(* IEC 61131-3 sources: AXOpen/src/components.keyence.vision/ctrl/src/Axo_IV3, 1 file *)

(* ---- Axo_IV3.st ---- *)
USING AXOpen.Core;
USING AXOpen.Messaging;
USING AXOpen.Messaging.Static;
USING AXOpen.Components.Abstractions;
USING Siemens.Simatic.Hardware.Utilities;

NAMESPACE AXOpen.Components.Keyence.Vision
    {S7.extern=ReadWrite}
    {#ix-prop: public string DeviceIpAddress}
    {#ix-prop: public string Proxy}
    CLASS Axo_IV3 EXTENDS AXOpen.Core.AxoComponent
        VAR PUBLIC // HEADER
            {#ix-attr:[Container(Layout.Wrap)]}
            {#ix-attr:[ComponentHeader()]}
            {#ix-set:AttributeName = "<#Progress#>"}
            Progress : INT;
        END_VAR

        VAR PUBLIC // TASKS
            {#ix-attr:[Container(Layout.Wrap)]}
            {#ix-attr:[ComponentDetails("Tasks")]}
            {#ix-set:AttributeName = "<#TriggerTask#>"}
            TriggerTask : AXOpen.Core.AxoTask;
            {#ix-attr:[Container(Layout.Wrap)]}
            {#ix-attr:[ComponentDetails("Tasks")]}
            {#ix-set:AttributeName = "<#Restore#>"}
            RestoreTask : AXOpen.Core.AxoTask;

            {#ix-attr:[Group(GroupLayout.GroupBox)]}
            {#ix-attr:[ComponentDetails("Tasks")]}
            {#ix-set:AttributeName = "<#Required program number#>"}
            RequiredProgramNumber : UINT;
            {#ix-attr:[ComponentDetails("Tasks")]}
            {#ix-set:AttributeName = "<#ChangeProgramTask#>"}
            ChangeProgramTask : AXOpen.Core.AxoTask;
        END_VAR

        VAR PUBLIC // CONFIG
            {#ix-attr:[Container(Layout.Stack)]}
            {#ix-attr:[ComponentDetails("Config")]}
            {#ix-attr:[ReadOnly()]}
            Config  :   Axo_IV3_Config;
        END_VAR

        VAR PUBLIC // STATUS
            {#ix-attr:[Container(Layout.Stack)]}
            {#ix-attr:[ComponentDetails("Status")]}
            {#ix-attr:[ReadOnly()]}
            Status              :   Axo_IV3_Component_Status;
            Messenger           :   AXOpen.Messaging.Static.AxoMessenger;
            TaskMessenger       :   AXOpen.Messaging.Static.AxoMessenger;
        END_VAR

        VAR PUBLIC // HARDWARE SIGNALS
            {#ix-attr:[ComponentDetails("HARDWARE SIGNALS")]}
            {#ix-attr:[Container(Layout.Wrap)]}
            {#ix-attr:[Group(GroupLayout.GroupBox)]}
            {#ix-set:AttributeName = "<#Inputs#>"}
            {#ix-attr:[ReadOnly()]}
            Inputs              :  Axo_IV3_In;
            {#ix-attr:[ComponentDetails("HARDWARE SIGNALS")]}
            {#ix-attr:[Container(Layout.Wrap)]}
            {#ix-attr:[Group(GroupLayout.GroupBox)]}
            {#ix-set:AttributeName = "<#Outputs#>"}
            {#ix-attr:[ReadOnly()]}
            Outputs              :   Axo_IV3_Out;
        END_VAR

        VAR PUBLIC // HARDWARE DIAGNOSTICS TASK
            {#ix-attr:[Container(Layout.Stack)]}
            {#ix-attr:[ComponentDetails("Hardware diagnostics")]}
            {#ix-set:AttributeName = "<#Update diagnostics#>"}
            HardwareDiagnosticsTask :   AXOpen.Io.AxoHardwareDiagnostics;

            LastProgressRoot : ARRAY[0..20] OF INT;
            ProgressRoot : ARRAY[0..20] OF INT;
            ActiveProgressRootIndex : INT;
        END_VAR

        VAR PRIVATE
            _progress       :   INT;
            _infoTimer      :   AXOpen.Timers.OnDelayTimer;
            _errorTimer     :   AXOpen.Timers.OnDelayTimer;
            _data_in        :   ARRAY[0..27] OF BYTE;
            _data_out_12    :   ARRAY[0..11] OF BYTE;
            _word           :   WORD;
            _dword          :   DWORD;

            _initHwCheckDone        :   BOOL;
            _retval                 :   WORD;
            _geoAddr                :   GeoAddr;
            _outHwid                :   UINT;
            _blink                  :   AXOpen.Timers.AxoBlinker;
            _inputsAddress          :   UDINT;
            _inputsCount            :   UINT;
            _outputsAddress         :   UDINT;
            _outputsCount           :   UINT;
            _resultUpdateComplete   :   BOOL;
            _resultNo               :   UINT;
            _programNumber          :   UINT;
            _ProgChangeInterrupted  :   BOOL;
        END_VAR

        METHOD AddProgressToRoot
            VAR_INPUT
                inProgress : INT;
            END_VAR

            var
                lastProgress : INT;
            end_var;

            lastProgress := ProgressRoot[ActiveProgressRootIndex];

            IF inProgress <> lastProgress THEN
                ActiveProgressRootIndex := ActiveProgressRootIndex + 1;
                IF ActiveProgressRootIndex > 20 THEN
                    ActiveProgressRootIndex := 0;
                END_IF;
                ProgressRoot[ActiveProgressRootIndex] := inProgress;
            END_IF;

        END_METHOD

        METHOD ClearProgressRoot
           var
            iterator : INT;
           end_var;

           ActiveProgressRootIndex := 0;
           FOR iterator := 0 TO 20 DO
            LastProgressRoot[iterator] := ProgressRoot[iterator];
                ProgressRoot[iterator] := -1;
           END_FOR;
        END_METHOD

        ///<summary>
        /// Runs tasks and logic of this component.
        /// >[!IMPORTANT] This method must or one of its overloads be called cyclically.
        ///</summary>
        METHOD PUBLIC Run
            VAR_INPUT
                inParent      :   IAxoObject;
                hwID        :   UINT;
            END_VAR

            SUPER.Run(inParent);

            Messenger.Serve(THIS);

            Progress := _progress;

            IF NOT _initHwCheckDone THEN
                IF inParent = NULL THEN
                    Messenger.Activate(UINT#700, eAxoMessageCategory#ProgrammingError);
                    Status.Error.Id := UINT#700;
                    RETURN;
                END_IF;
                IF hwID = UINT#0 THEN
                    Messenger.Activate(UINT#701, eAxoMessageCategory#ProgrammingError);
                    Status.Error.Id := UINT#701;
                    RETURN;
                END_IF;

                Config.HWIDs.HW_Device := hwID;
                _retval := ReadSlotFromHardwareID(hardwareID := Config.HWIDs.HW_Device, geoAddr :=_geoAddr);
                IF _retval = WORD#8090 THEN
                    Messenger.Activate(UINT#702,eAxoMessageCategory#Error);
                    Status.Error.Id := UINT#702;
                    RETURN;
                END_IF;

                //******************Slot 1*****************//
                _geoAddr.Slot   :=  UINT#1;
                _geoAddr.HardwareType := UINT#4; // (4-Module)
                _retval := ReadHardwareIDFromSlot(geoAddr := _geoAddr, hardwareID => Config.HWIDs.HwID_CommandControl);
                IF Config.HWIDs.HwID_CommandControl = UINT#0 THEN
                    Messenger.Activate(UINT#710,eAxoMessageCategory#Error);
                    Status.Error.Id := UINT#710;
                    RETURN;
                END_IF;
                IF _retval = WORD#8091 THEN
                    Messenger.Activate(UINT#711,eAxoMessageCategory#Error);
                    Status.Error.Id := UINT#711;
                    RETURN;
                END_IF;
                IF _retval = WORD#8094 THEN
                    Messenger.Activate(UINT#712,eAxoMessageCategory#Error);
                    Status.Error.Id := UINT#712;
                    RETURN;
                END_IF;
                IF _retval = WORD#8095 THEN
                    Messenger.Activate(UINT#713,eAxoMessageCategory#Error);
                    Status.Error.Id := UINT#713;
                    RETURN;
                END_IF;
                IF _retval = WORD#8096 THEN
                    Messenger.Activate(UINT#714,eAxoMessageCategory#Error);
                    Status.Error.Id := UINT#714;
                    RETURN;
                END_IF;
                IF _retval = WORD#8097 THEN
                    Messenger.Activate(UINT#715,eAxoMessageCategory#Error);
                    Status.Error.Id := UINT#715;
                    RETURN;
                END_IF;
                ReadHardwareIOAddress(hardwareID := (Config.HWIDs.HwID_CommandControl) , inputStartAddress => _inputsAddress , inputCount => _inputsCount , outputStartAddress => _outputsAddress , outputCount => _outputsCount);
                IF _inputsCount <> UINT#0 OR _outputsCount <> UINT#12 THEN
                    Messenger.Activate(UINT#716,eAxoMessageCategory#Error);
                    Status.Error.Id := UINT#716;
                    RETURN;
                END_IF;
                //******************Slot 2*****************//
                _geoAddr.Slot   :=  UINT#2;
                _geoAddr.HardwareType := UINT#4; // (4-Module)
                _retval := ReadHardwareIDFromSlot(geoAddr := _geoAddr, hardwareID => Config.HWIDs.HwID_CommandStatusBits);
                IF Config.HWIDs.HwID_CommandStatusBits = UINT#0 THEN
                    Messenger.Activate(UINT#720,eAxoMessageCategory#Error);
                    Status.Error.Id := UINT#720;
                    RETURN;
                END_IF;
                IF _retval = WORD#8091 THEN
                    Messenger.Activate(UINT#721,eAxoMessageCategory#Error);
                    Status.Error.Id := UINT#721;
                    RETURN;
                END_IF;
                IF _retval = WORD#8094 THEN
                    Messenger.Activate(UINT#722,eAxoMessageCategory#Error);
                    Status.Error.Id := UINT#722;
                    RETURN;
                END_IF;
                IF _retval = WORD#8095 THEN
                    Messenger.Activate(UINT#723,eAxoMessageCategory#Error);
                    Status.Error.Id := UINT#723;
                    RETURN;
                END_IF;
                IF _retval = WORD#8096 THEN
                    Messenger.Activate(UINT#724,eAxoMessageCategory#Error);
                    Status.Error.Id := UINT#724;
                    RETURN;
                END_IF;
                IF _retval = WORD#8097 THEN
                    Messenger.Activate(UINT#725,eAxoMessageCategory#Error);
                    Status.Error.Id := UINT#725;
                    RETURN;
                END_IF;
                ReadHardwareIOAddress(hardwareID := (Config.HWIDs.HwID_CommandStatusBits) , inputStartAddress => _inputsAddress , inputCount => _inputsCount , outputStartAddress => _outputsAddress , outputCount => _outputsCount);
                IF _inputsCount <> UINT#4 OR _outputsCount <> UINT#0 THEN
                    Messenger.Activate(UINT#726,eAxoMessageCategory#Error);
                    Status.Error.Id := UINT#726;
                    RETURN;
                END_IF;
                //******************Slot 3*****************//
                _geoAddr.Slot   :=  UINT#3;
                _geoAddr.HardwareType := UINT#4; // (4-Module)
                _retval := ReadHardwareIDFromSlot(geoAddr := _geoAddr, hardwareID => Config.HWIDs.HwID_DeviceResultBits_1);
                IF Config.HWIDs.HwID_DeviceResultBits_1 = UINT#0 THEN
                    Messenger.Activate(UINT#730,eAxoMessageCategory#Error);
                    Status.Error.Id := UINT#730;
                    RETURN;
                END_IF;
                IF _retval = WORD#8091 THEN
                    Messenger.Activate(UINT#731,eAxoMessageCategory#Error);
                    Status.Error.Id := UINT#731;
                    RETURN;
                END_IF;
                IF _retval = WORD#8094 THEN
                    Messenger.Activate(UINT#732,eAxoMessageCategory#Error);
                    Status.Error.Id := UINT#732;
                    RETURN;
                END_IF;
                IF _retval = WORD#8095 THEN
                    Messenger.Activate(UINT#733,eAxoMessageCategory#Error);
                    Status.Error.Id := UINT#733;
                    RETURN;
                END_IF;
                IF _retval = WORD#8096 THEN
                    Messenger.Activate(UINT#734,eAxoMessageCategory#Error);
                    Status.Error.Id := UINT#734;
                    RETURN;
                END_IF;
                IF _retval = WORD#8097 THEN
                    Messenger.Activate(UINT#735,eAxoMessageCategory#Error);
                    Status.Error.Id := UINT#735;
                    RETURN;
                END_IF;
                ReadHardwareIOAddress(hardwareID := (Config.HWIDs.HwID_DeviceResultBits_1) , inputStartAddress => _inputsAddress , inputCount => _inputsCount , outputStartAddress => _outputsAddress , outputCount => _outputsCount);
                IF _inputsCount <> UINT#4 OR _outputsCount <> UINT#0 THEN
                    Messenger.Activate(UINT#736,eAxoMessageCategory#Error);
                    Status.Error.Id := UINT#736;
                    RETURN;
                END_IF;
                //******************Slot 4*****************//
                _geoAddr.Slot   :=  UINT#4;
                _geoAddr.HardwareType := UINT#4; // (4-Module)
                _retval := ReadHardwareIDFromSlot(geoAddr := _geoAddr, hardwareID => Config.HWIDs.HwID_DeviceStatusWords);
                IF Config.HWIDs.HwID_DeviceStatusWords = UINT#0 THEN
                    Messenger.Activate(UINT#740,eAxoMessageCategory#Error);
                    Status.Error.Id := UINT#740;
                    RETURN;
                END_IF;
                IF _retval = WORD#8091 THEN
                    Messenger.Activate(UINT#741,eAxoMessageCategory#Error);
                    Status.Error.Id := UINT#741;
                    RETURN;
                END_IF;
                IF _retval = WORD#8094 THEN
                    Messenger.Activate(UINT#742,eAxoMessageCategory#Error);
                    Status.Error.Id := UINT#742;
                    RETURN;
                END_IF;
                IF _retval = WORD#8095 THEN
                    Messenger.Activate(UINT#743,eAxoMessageCategory#Error);
                    Status.Error.Id := UINT#743;
                    RETURN;
                END_IF;
                IF _retval = WORD#8096 THEN
                    Messenger.Activate(UINT#744,eAxoMessageCategory#Error);
                    Status.Error.Id := UINT#744;
                    RETURN;
                END_IF;
                IF _retval = WORD#8097 THEN
                    Messenger.Activate(UINT#745,eAxoMessageCategory#Error);
                    Status.Error.Id := UINT#745;
                    RETURN;
                END_IF;
                ReadHardwareIOAddress(hardwareID := (Config.HWIDs.HwID_DeviceStatusWords) , inputStartAddress => _inputsAddress , inputCount => _inputsCount , outputStartAddress => _outputsAddress , outputCount => _outputsCount);
                IF _inputsCount <> UINT#16 OR _outputsCount <> UINT#0 THEN
                    Messenger.Activate(UINT#746,eAxoMessageCategory#Error);
                    Status.Error.Id := UINT#746;
                    RETURN;
                END_IF;
                //******************Slot 5*****************//
                _geoAddr.Slot   :=  UINT#5;
                _geoAddr.HardwareType := UINT#4; // (4-Module)
                _retval := ReadHardwareIDFromSlot(geoAddr := _geoAddr, hardwareID => Config.HWIDs.HwID_DeviceStatistics);
                IF Config.HWIDs.HwID_DeviceStatistics = UINT#0 THEN
                    Messenger.Activate(UINT#750,eAxoMessageCategory#Error);
                    Status.Error.Id := UINT#750;
                    RETURN;
                END_IF;
                IF _retval = WORD#8091 THEN
                    Messenger.Activate(UINT#751,eAxoMessageCategory#Error);
                    Status.Error.Id := UINT#751;
                    RETURN;
                END_IF;
                IF _retval = WORD#8094 THEN
                    Messenger.Activate(UINT#752,eAxoMessageCategory#Error);
                    Status.Error.Id := UINT#752;
                    RETURN;
                END_IF;
                IF _retval = WORD#8095 THEN
                    Messenger.Activate(UINT#753,eAxoMessageCategory#Error);
                    Status.Error.Id := UINT#753;
                    RETURN;
                END_IF;
                IF _retval = WORD#8096 THEN
                    Messenger.Activate(UINT#754,eAxoMessageCategory#Error);
                    Status.Error.Id := UINT#754;
                    RETURN;
                END_IF;
                IF _retval = WORD#8097 THEN
                    Messenger.Activate(UINT#755,eAxoMessageCategory#Error);
                    Status.Error.Id := UINT#755;
                    RETURN;
                END_IF;
                ReadHardwareIOAddress(hardwareID := (Config.HWIDs.HwID_DeviceStatistics) , inputStartAddress => _inputsAddress , inputCount => _inputsCount , outputStartAddress => _outputsAddress , outputCount => _outputsCount);
                IF _inputsCount <> UINT#28 OR _outputsCount <> UINT#0 THEN
                    Messenger.Activate(UINT#756,eAxoMessageCategory#Error);
                    Status.Error.Id := UINT#756;
                    RETURN;
                END_IF;
                //******************Slot 6*****************//
                _geoAddr.Slot   :=  UINT#6;
                _geoAddr.HardwareType := UINT#4; // (4-Module)
                _retval := ReadHardwareIDFromSlot(geoAddr := _geoAddr, hardwareID => Config.HWIDs.HwID_PositionAdjustResult);
                IF Config.HWIDs.HwID_PositionAdjustResult = UINT#0 THEN
                    Messenger.Activate(UINT#760,eAxoMessageCategory#Error);
                    Status.Error.Id := UINT#760;
                    RETURN;
                END_IF;
                IF _retval = WORD#8091 THEN
                    Messenger.Activate(UINT#761,eAxoMessageCategory#Error);
                    Status.Error.Id := UINT#761;
                    RETURN;
                END_IF;
                IF _retval = WORD#8094 THEN
                    Messenger.Activate(UINT#762,eAxoMessageCategory#Error);
                    Status.Error.Id := UINT#762;
                    RETURN;
                END_IF;
                IF _retval = WORD#8095 THEN
                    Messenger.Activate(UINT#763,eAxoMessageCategory#Error);
                    Status.Error.Id := UINT#763;
                    RETURN;
                END_IF;
                IF _retval = WORD#8096 THEN
                    Messenger.Activate(UINT#764,eAxoMessageCategory#Error);
                    Status.Error.Id := UINT#764;
                    RETURN;
                END_IF;
                IF _retval = WORD#8097 THEN
                    Messenger.Activate(UINT#765,eAxoMessageCategory#Error);
                    Status.Error.Id := UINT#765;
                    RETURN;
                END_IF;
                ReadHardwareIOAddress(hardwareID := (Config.HWIDs.HwID_PositionAdjustResult) , inputStartAddress => _inputsAddress , inputCount => _inputsCount , outputStartAddress => _outputsAddress , outputCount => _outputsCount);
                IF _inputsCount <> UINT#20 OR _outputsCount <> UINT#0 THEN
                    Messenger.Activate(UINT#766,eAxoMessageCategory#Error);
                    Status.Error.Id := UINT#766;
                    RETURN;
                END_IF;
                //******************Slot 7*****************//
                _geoAddr.Slot   :=  UINT#7;
                _geoAddr.HardwareType := UINT#4; // (4-Module)
                _retval := ReadHardwareIDFromSlot(geoAddr := _geoAddr, hardwareID => Config.HWIDs.HwID_ToolResult_1);
                IF Config.HWIDs.HwID_ToolResult_1 = UINT#0 THEN
                    Messenger.Activate(UINT#770,eAxoMessageCategory#Error);
                    Status.Error.Id := UINT#770;
                    RETURN;
                END_IF;
                IF _retval = WORD#8091 THEN
                    Messenger.Activate(UINT#771,eAxoMessageCategory#Error);
                    Status.Error.Id := UINT#771;
                    RETURN;
                END_IF;
                IF _retval = WORD#8094 THEN
                    Messenger.Activate(UINT#772,eAxoMessageCategory#Error);
                    Status.Error.Id := UINT#772;
                    RETURN;
                END_IF;
                IF _retval = WORD#8095 THEN
                    Messenger.Activate(UINT#773,eAxoMessageCategory#Error);
                    Status.Error.Id := UINT#773;
                    RETURN;
                END_IF;
                IF _retval = WORD#8096 THEN
                    Messenger.Activate(UINT#774,eAxoMessageCategory#Error);
                    Status.Error.Id := UINT#774;
                    RETURN;
                END_IF;
                IF _retval = WORD#8097 THEN
                    Messenger.Activate(UINT#775,eAxoMessageCategory#Error);
                    Status.Error.Id := UINT#775;
                    RETURN;
                END_IF;
                ReadHardwareIOAddress(hardwareID := (Config.HWIDs.HwID_ToolResult_1) , inputStartAddress => _inputsAddress , inputCount => _inputsCount , outputStartAddress => _outputsAddress , outputCount => _outputsCount);
                IF _inputsCount <> UINT#20 OR _outputsCount <> UINT#0 THEN
                    Messenger.Activate(UINT#776,eAxoMessageCategory#Error);
                    Status.Error.Id := UINT#776;
                    RETURN;
                END_IF;
                //******************Slot 8*****************//
                _geoAddr.Slot   :=  UINT#8;
                _geoAddr.HardwareType := UINT#4; // (4-Module)
                _retval := ReadHardwareIDFromSlot(geoAddr := _geoAddr, hardwareID => Config.HWIDs.HwID_ToolResult_2);
                IF Config.HWIDs.HwID_ToolResult_2 = UINT#0 THEN
                    Messenger.Activate(UINT#780,eAxoMessageCategory#Error);
                    Status.Error.Id := UINT#780;
                    RETURN;
                END_IF;
                IF _retval = WORD#8091 THEN
                    Messenger.Activate(UINT#781,eAxoMessageCategory#Error);
                    Status.Error.Id := UINT#781;
                    RETURN;
                END_IF;
                IF _retval = WORD#8094 THEN
                    Messenger.Activate(UINT#782,eAxoMessageCategory#Error);
                    Status.Error.Id := UINT#782;
                    RETURN;
                END_IF;
                IF _retval = WORD#8095 THEN
                    Messenger.Activate(UINT#783,eAxoMessageCategory#Error);
                    Status.Error.Id := UINT#783;
                    RETURN;
                END_IF;
                IF _retval = WORD#8096 THEN
                    Messenger.Activate(UINT#784,eAxoMessageCategory#Error);
                    Status.Error.Id := UINT#784;
                    RETURN;
                END_IF;
                IF _retval = WORD#8097 THEN
                    Messenger.Activate(UINT#785,eAxoMessageCategory#Error);
                    Status.Error.Id := UINT#785;
                    RETURN;
                END_IF;
                ReadHardwareIOAddress(hardwareID := (Config.HWIDs.HwID_ToolResult_2) , inputStartAddress => _inputsAddress , inputCount => _inputsCount , outputStartAddress => _outputsAddress , outputCount => _outputsCount);
                IF _inputsCount <> UINT#20 OR _outputsCount <> UINT#0 THEN
                    Messenger.Activate(UINT#786,eAxoMessageCategory#Error);
                    Status.Error.Id := UINT#786;
                    RETURN;
                END_IF;
                //******************Slot 9*****************//
                _geoAddr.Slot   :=  UINT#9;
                _geoAddr.HardwareType := UINT#4; // (4-Module)
                _retval := ReadHardwareIDFromSlot(geoAddr := _geoAddr, hardwareID => Config.HWIDs.HwID_ToolResult_3);
                IF Config.HWIDs.HwID_ToolResult_3 = UINT#0 THEN
                    Messenger.Activate(UINT#790,eAxoMessageCategory#Error);
                    Status.Error.Id := UINT#790;
                    RETURN;
                END_IF;
                IF _retval = WORD#8091 THEN
                    Messenger.Activate(UINT#791,eAxoMessageCategory#Error);
                    Status.Error.Id := UINT#791;
                    RETURN;
                END_IF;
                IF _retval = WORD#8094 THEN
                    Messenger.Activate(UINT#792,eAxoMessageCategory#Error);
                    Status.Error.Id := UINT#792;
                    RETURN;
                END_IF;
                IF _retval = WORD#8095 THEN
                    Messenger.Activate(UINT#793,eAxoMessageCategory#Error);
                    Status.Error.Id := UINT#793;
                    RETURN;
                END_IF;
                IF _retval = WORD#8096 THEN
                    Messenger.Activate(UINT#794,eAxoMessageCategory#Error);
                    Status.Error.Id := UINT#794;
                    RETURN;
                END_IF;
                IF _retval = WORD#8097 THEN
                    Messenger.Activate(UINT#795,eAxoMessageCategory#Error);
                    Status.Error.Id := UINT#795;
                    RETURN;
                END_IF;
                ReadHardwareIOAddress(hardwareID := (Config.HWIDs.HwID_ToolResult_3) , inputStartAddress => _inputsAddress , inputCount => _inputsCount , outputStartAddress => _outputsAddress , outputCount => _outputsCount);
                IF _inputsCount <> UINT#20 OR _outputsCount <> UINT#0 THEN
                    Messenger.Activate(UINT#796,eAxoMessageCategory#Error);
                    Status.Error.Id := UINT#796;
                    RETURN;
                END_IF;
                //******************Slot 10*****************//
                _geoAddr.Slot   :=  UINT#10;
                _geoAddr.HardwareType := UINT#4; // (4-Module)
                _retval := ReadHardwareIDFromSlot(geoAddr := _geoAddr, hardwareID => Config.HWIDs.HwID_ToolResult_4);
                IF Config.HWIDs.HwID_ToolResult_4 = UINT#0 THEN
                    Messenger.Activate(UINT#800,eAxoMessageCategory#Error);
                    Status.Error.Id := UINT#800;
                    RETURN;
                END_IF;
                IF _retval = WORD#8091 THEN
                    Messenger.Activate(UINT#801,eAxoMessageCategory#Error);
                    Status.Error.Id := UINT#801;
                    RETURN;
                END_IF;
                IF _retval = WORD#8094 THEN
                    Messenger.Activate(UINT#802,eAxoMessageCategory#Error);
                    Status.Error.Id := UINT#802;
                    RETURN;
                END_IF;
                IF _retval = WORD#8095 THEN
                    Messenger.Activate(UINT#803,eAxoMessageCategory#Error);
                    Status.Error.Id := UINT#803;
                    RETURN;
                END_IF;
                IF _retval = WORD#8096 THEN
                    Messenger.Activate(UINT#804,eAxoMessageCategory#Error);
                    Status.Error.Id := UINT#804;
                    RETURN;
                END_IF;
                IF _retval = WORD#8097 THEN
                    Messenger.Activate(UINT#805,eAxoMessageCategory#Error);
                    Status.Error.Id := UINT#805;
                    RETURN;
                END_IF;
                ReadHardwareIOAddress(hardwareID := (Config.HWIDs.HwID_ToolResult_4) , inputStartAddress => _inputsAddress , inputCount => _inputsCount , outputStartAddress => _outputsAddress , outputCount => _outputsCount);
                IF _inputsCount <> UINT#20 OR _outputsCount <> UINT#0 THEN
                    Messenger.Activate(UINT#806,eAxoMessageCategory#Error);
                    Status.Error.Id := UINT#806;
                    RETURN;
                END_IF;
                //******************Slot 11*****************//
                _geoAddr.Slot   :=  UINT#11;
                _geoAddr.HardwareType := UINT#4; // (4-Module)
                _retval := ReadHardwareIDFromSlot(geoAddr := _geoAddr, hardwareID => Config.HWIDs.HwID_ToolResult_5);
                IF Config.HWIDs.HwID_ToolResult_5 = UINT#0 THEN
                    Messenger.Activate(UINT#810,eAxoMessageCategory#Error);
                    Status.Error.Id := UINT#810;
                    RETURN;
                END_IF;
                IF _retval = WORD#8091 THEN
                    Messenger.Activate(UINT#811,eAxoMessageCategory#Error);
                    Status.Error.Id := UINT#811;
                    RETURN;
                END_IF;
                IF _retval = WORD#8094 THEN
                    Messenger.Activate(UINT#812,eAxoMessageCategory#Error);
                    Status.Error.Id := UINT#812;
                    RETURN;
                END_IF;
                IF _retval = WORD#8095 THEN
                    Messenger.Activate(UINT#813,eAxoMessageCategory#Error);
                    Status.Error.Id := UINT#813;
                    RETURN;
                END_IF;
                IF _retval = WORD#8096 THEN
                    Messenger.Activate(UINT#814,eAxoMessageCategory#Error);
                    Status.Error.Id := UINT#814;
                    RETURN;
                END_IF;
                IF _retval = WORD#8097 THEN
                    Messenger.Activate(UINT#815,eAxoMessageCategory#Error);
                    Status.Error.Id := UINT#815;
                    RETURN;
                END_IF;
                ReadHardwareIOAddress(hardwareID := (Config.HWIDs.HwID_ToolResult_5) , inputStartAddress => _inputsAddress , inputCount => _inputsCount , outputStartAddress => _outputsAddress , outputCount => _outputsCount);
                IF _inputsCount <> UINT#20 OR _outputsCount <> UINT#0 THEN
                    Messenger.Activate(UINT#816,eAxoMessageCategory#Error);
                    Status.Error.Id := UINT#816;
                    RETURN;
                END_IF;
                //******************Slot 12*****************//
                _geoAddr.Slot   :=  UINT#12;
                _geoAddr.HardwareType := UINT#4; // (4-Module)
                _retval := ReadHardwareIDFromSlot(geoAddr := _geoAddr, hardwareID => Config.HWIDs.HwID_ToolResult_6);
                IF Config.HWIDs.HwID_ToolResult_6 = UINT#0 THEN
                    Messenger.Activate(UINT#820,eAxoMessageCategory#Error);
                    Status.Error.Id := UINT#820;
                    RETURN;
                END_IF;
                IF _retval = WORD#8091 THEN
                    Messenger.Activate(UINT#821,eAxoMessageCategory#Error);
                    Status.Error.Id := UINT#821;
                    RETURN;
                END_IF;
                IF _retval = WORD#8094 THEN
                    Messenger.Activate(UINT#822,eAxoMessageCategory#Error);
                    Status.Error.Id := UINT#822;
                    RETURN;
                END_IF;
                IF _retval = WORD#8095 THEN
                    Messenger.Activate(UINT#823,eAxoMessageCategory#Error);
                    Status.Error.Id := UINT#823;
                    RETURN;
                END_IF;
                IF _retval = WORD#8096 THEN
                    Messenger.Activate(UINT#824,eAxoMessageCategory#Error);
                    Status.Error.Id := UINT#824;
                    RETURN;
                END_IF;
                IF _retval = WORD#8097 THEN
                    Messenger.Activate(UINT#825,eAxoMessageCategory#Error);
                    Status.Error.Id := UINT#825;
                    RETURN;
                END_IF;
                ReadHardwareIOAddress(hardwareID := (Config.HWIDs.HwID_ToolResult_6) , inputStartAddress => _inputsAddress , inputCount => _inputsCount , outputStartAddress => _outputsAddress , outputCount => _outputsCount);
                IF _inputsCount <> UINT#20 OR _outputsCount <> UINT#0 THEN
                    Messenger.Activate(UINT#826,eAxoMessageCategory#Error);
                    Status.Error.Id := UINT#826;
                    RETURN;
                END_IF;
                //******************Slot 13*****************//
                _geoAddr.Slot   :=  UINT#13;
                _geoAddr.HardwareType := UINT#4; // (4-Module)
                _retval := ReadHardwareIDFromSlot(geoAddr := _geoAddr, hardwareID => Config.HWIDs.HwID_ToolResult_7);
                IF Config.HWIDs.HwID_ToolResult_7 = UINT#0 THEN
                    Messenger.Activate(UINT#830,eAxoMessageCategory#Error);
                    Status.Error.Id := UINT#830;
                    RETURN;
                END_IF;
                IF _retval = WORD#8091 THEN
                    Messenger.Activate(UINT#831,eAxoMessageCategory#Error);
                    Status.Error.Id := UINT#831;
                    RETURN;
                END_IF;
                IF _retval = WORD#8094 THEN
                    Messenger.Activate(UINT#832,eAxoMessageCategory#Error);
                    Status.Error.Id := UINT#832;
                    RETURN;
                END_IF;
                IF _retval = WORD#8095 THEN
                    Messenger.Activate(UINT#833,eAxoMessageCategory#Error);
                    Status.Error.Id := UINT#833;
                    RETURN;
                END_IF;
                IF _retval = WORD#8096 THEN
                    Messenger.Activate(UINT#834,eAxoMessageCategory#Error);
                    Status.Error.Id := UINT#834;
                    RETURN;
                END_IF;
                IF _retval = WORD#8097 THEN
                    Messenger.Activate(UINT#835,eAxoMessageCategory#Error);
                    Status.Error.Id := UINT#835;
                    RETURN;
                END_IF;
                ReadHardwareIOAddress(hardwareID := (Config.HWIDs.HwID_ToolResult_7) , inputStartAddress => _inputsAddress , inputCount => _inputsCount , outputStartAddress => _outputsAddress , outputCount => _outputsCount);
                IF _inputsCount <> UINT#20 OR _outputsCount <> UINT#0 THEN
                    Messenger.Activate(UINT#836,eAxoMessageCategory#Error);
                    Status.Error.Id := UINT#836;
                    RETURN;
                END_IF;
                //******************Slot 14*****************//
                _geoAddr.Slot   :=  UINT#14;
                _geoAddr.HardwareType := UINT#4; // (4-Module)
                _retval := ReadHardwareIDFromSlot(geoAddr := _geoAddr, hardwareID => Config.HWIDs.HwID_ToolResult_8);
                IF Config.HWIDs.HwID_ToolResult_8 = UINT#0 THEN
                    Messenger.Activate(UINT#840,eAxoMessageCategory#Error);
                    Status.Error.Id := UINT#840;
                    RETURN;
                END_IF;
                IF _retval = WORD#8091 THEN
                    Messenger.Activate(UINT#841,eAxoMessageCategory#Error);
                    Status.Error.Id := UINT#841;
                    RETURN;
                END_IF;
                IF _retval = WORD#8094 THEN
                    Messenger.Activate(UINT#842,eAxoMessageCategory#Error);
                    Status.Error.Id := UINT#842;
                    RETURN;
                END_IF;
                IF _retval = WORD#8095 THEN
                    Messenger.Activate(UINT#843,eAxoMessageCategory#Error);
                    Status.Error.Id := UINT#843;
                    RETURN;
                END_IF;
                IF _retval = WORD#8096 THEN
                    Messenger.Activate(UINT#844,eAxoMessageCategory#Error);
                    Status.Error.Id := UINT#844;
                    RETURN;
                END_IF;
                IF _retval = WORD#8097 THEN
                    Messenger.Activate(UINT#845,eAxoMessageCategory#Error);
                    Status.Error.Id := UINT#845;
                    RETURN;
                END_IF;
                ReadHardwareIOAddress(hardwareID := (Config.HWIDs.HwID_ToolResult_8) , inputStartAddress => _inputsAddress , inputCount => _inputsCount , outputStartAddress => _outputsAddress , outputCount => _outputsCount);
                IF _inputsCount <> UINT#20 OR _outputsCount <> UINT#0 THEN
                    Messenger.Activate(UINT#846,eAxoMessageCategory#Error);
                    Status.Error.Id := UINT#846;
                    RETURN;
                END_IF;
                //******************Slot 15*****************//
                _geoAddr.Slot   :=  UINT#15;
                _geoAddr.HardwareType := UINT#4; // (4-Module)
                _retval := ReadHardwareIDFromSlot(geoAddr := _geoAddr, hardwareID => Config.HWIDs.HwID_ToolResult_9);
                IF Config.HWIDs.HwID_ToolResult_9 = UINT#0 THEN
                    Messenger.Activate(UINT#850,eAxoMessageCategory#Error);
                    Status.Error.Id := UINT#850;
                    RETURN;
                END_IF;
                IF _retval = WORD#8091 THEN
                    Messenger.Activate(UINT#851,eAxoMessageCategory#Error);
                    Status.Error.Id := UINT#851;
                    RETURN;
                END_IF;
                IF _retval = WORD#8094 THEN
                    Messenger.Activate(UINT#852,eAxoMessageCategory#Error);
                    Status.Error.Id := UINT#852;
                    RETURN;
                END_IF;
                IF _retval = WORD#8095 THEN
                    Messenger.Activate(UINT#853,eAxoMessageCategory#Error);
                    Status.Error.Id := UINT#853;
                    RETURN;
                END_IF;
                IF _retval = WORD#8096 THEN
                    Messenger.Activate(UINT#854,eAxoMessageCategory#Error);
                    Status.Error.Id := UINT#854;
                    RETURN;
                END_IF;
                IF _retval = WORD#8097 THEN
                    Messenger.Activate(UINT#855,eAxoMessageCategory#Error);
                    Status.Error.Id := UINT#855;
                    RETURN;
                END_IF;
                ReadHardwareIOAddress(hardwareID := (Config.HWIDs.HwID_ToolResult_9) , inputStartAddress => _inputsAddress , inputCount => _inputsCount , outputStartAddress => _outputsAddress , outputCount => _outputsCount);
                IF _inputsCount <> UINT#20 OR _outputsCount <> UINT#0 THEN
                    Messenger.Activate(UINT#856,eAxoMessageCategory#Error);
                    Status.Error.Id := UINT#856;
                    RETURN;
                END_IF;
                //******************Slot 16*****************//
                _geoAddr.Slot   :=  UINT#16;
                _geoAddr.HardwareType := UINT#4; // (4-Module)
                _retval := ReadHardwareIDFromSlot(geoAddr := _geoAddr, hardwareID => Config.HWIDs.HwID_ToolResult_10);
                IF Config.HWIDs.HwID_ToolResult_10 = UINT#0 THEN
                    Messenger.Activate(UINT#860,eAxoMessageCategory#Error);
                    Status.Error.Id := UINT#860;
                    RETURN;
                END_IF;
                IF _retval = WORD#8091 THEN
                    Messenger.Activate(UINT#861,eAxoMessageCategory#Error);
                    Status.Error.Id := UINT#861;
                    RETURN;
                END_IF;
                IF _retval = WORD#8094 THEN
                    Messenger.Activate(UINT#862,eAxoMessageCategory#Error);
                    Status.Error.Id := UINT#862;
                    RETURN;
                END_IF;
                IF _retval = WORD#8095 THEN
                    Messenger.Activate(UINT#863,eAxoMessageCategory#Error);
                    Status.Error.Id := UINT#863;
                    RETURN;
                END_IF;
                IF _retval = WORD#8096 THEN
                    Messenger.Activate(UINT#864,eAxoMessageCategory#Error);
                    Status.Error.Id := UINT#864;
                    RETURN;
                END_IF;
                IF _retval = WORD#8097 THEN
                    Messenger.Activate(UINT#865,eAxoMessageCategory#Error);
                    Status.Error.Id := UINT#865;
                    RETURN;
                END_IF;
                ReadHardwareIOAddress(hardwareID := (Config.HWIDs.HwID_ToolResult_10) , inputStartAddress => _inputsAddress , inputCount => _inputsCount , outputStartAddress => _outputsAddress , outputCount => _outputsCount);
                IF _inputsCount <> UINT#20 OR _outputsCount <> UINT#0 THEN
                    Messenger.Activate(UINT#866,eAxoMessageCategory#Error);
                    Status.Error.Id := UINT#866;
                    RETURN;
                END_IF;
                //******************Slot 17*****************//
                _geoAddr.Slot   :=  UINT#17;
                _geoAddr.HardwareType := UINT#4; // (4-Module)
                _retval := ReadHardwareIDFromSlot(geoAddr := _geoAddr, hardwareID => Config.HWIDs.HwID_ToolResult_11);
                IF Config.HWIDs.HwID_ToolResult_11 = UINT#0 THEN
                    Messenger.Activate(UINT#870,eAxoMessageCategory#Error);
                    Status.Error.Id := UINT#870;
                    RETURN;
                END_IF;
                IF _retval = WORD#8091 THEN
                    Messenger.Activate(UINT#871,eAxoMessageCategory#Error);
                    Status.Error.Id := UINT#871;
                    RETURN;
                END_IF;
                IF _retval = WORD#8094 THEN
                    Messenger.Activate(UINT#872,eAxoMessageCategory#Error);
                    Status.Error.Id := UINT#872;
                    RETURN;
                END_IF;
                IF _retval = WORD#8095 THEN
                    Messenger.Activate(UINT#873,eAxoMessageCategory#Error);
                    Status.Error.Id := UINT#873;
                    RETURN;
                END_IF;
                IF _retval = WORD#8096 THEN
                    Messenger.Activate(UINT#874,eAxoMessageCategory#Error);
                    Status.Error.Id := UINT#874;
                    RETURN;
                END_IF;
                IF _retval = WORD#8097 THEN
                    Messenger.Activate(UINT#875,eAxoMessageCategory#Error);
                    Status.Error.Id := UINT#875;
                    RETURN;
                END_IF;
                ReadHardwareIOAddress(hardwareID := (Config.HWIDs.HwID_ToolResult_11) , inputStartAddress => _inputsAddress , inputCount => _inputsCount , outputStartAddress => _outputsAddress , outputCount => _outputsCount);
                IF _inputsCount <> UINT#20 OR _outputsCount <> UINT#0 THEN
                    Messenger.Activate(UINT#876,eAxoMessageCategory#Error);
                    Status.Error.Id := UINT#876;
                    RETURN;
                END_IF;
                //******************Slot 18*****************//
                _geoAddr.Slot   :=  UINT#18;
                _geoAddr.HardwareType := UINT#4; // (4-Module)
                _retval := ReadHardwareIDFromSlot(geoAddr := _geoAddr, hardwareID => Config.HWIDs.HwID_ToolResult_12);
                IF Config.HWIDs.HwID_ToolResult_12 = UINT#0 THEN
                    Messenger.Activate(UINT#880,eAxoMessageCategory#Error);
                    Status.Error.Id := UINT#880;
                    RETURN;
                END_IF;
                IF _retval = WORD#8091 THEN
                    Messenger.Activate(UINT#881,eAxoMessageCategory#Error);
                    Status.Error.Id := UINT#881;
                    RETURN;
                END_IF;
                IF _retval = WORD#8094 THEN
                    Messenger.Activate(UINT#882,eAxoMessageCategory#Error);
                    Status.Error.Id := UINT#882;
                    RETURN;
                END_IF;
                IF _retval = WORD#8095 THEN
                    Messenger.Activate(UINT#883,eAxoMessageCategory#Error);
                    Status.Error.Id := UINT#883;
                    RETURN;
                END_IF;
                IF _retval = WORD#8096 THEN
                    Messenger.Activate(UINT#884,eAxoMessageCategory#Error);
                    Status.Error.Id := UINT#884;
                    RETURN;
                END_IF;
                IF _retval = WORD#8097 THEN
                    Messenger.Activate(UINT#885,eAxoMessageCategory#Error);
                    Status.Error.Id := UINT#885;
                    RETURN;
                END_IF;
                ReadHardwareIOAddress(hardwareID := (Config.HWIDs.HwID_ToolResult_12) , inputStartAddress => _inputsAddress , inputCount => _inputsCount , outputStartAddress => _outputsAddress , outputCount => _outputsCount);
                IF _inputsCount <> UINT#20 OR _outputsCount <> UINT#0 THEN
                    Messenger.Activate(UINT#886,eAxoMessageCategory#Error);
                    Status.Error.Id := UINT#886;
                    RETURN;
                END_IF;
                //******************Slot 19*****************//
                _geoAddr.Slot   :=  UINT#19;
                _geoAddr.HardwareType := UINT#4; // (4-Module)
                _retval := ReadHardwareIDFromSlot(geoAddr := _geoAddr, hardwareID => Config.HWIDs.HwID_ToolResult_13);
                IF Config.HWIDs.HwID_ToolResult_13 = UINT#0 THEN
                    Messenger.Activate(UINT#890,eAxoMessageCategory#Error);
                    Status.Error.Id := UINT#890;
                    RETURN;
                END_IF;
                IF _retval = WORD#8091 THEN
                    Messenger.Activate(UINT#891,eAxoMessageCategory#Error);
                    Status.Error.Id := UINT#891;
                    RETURN;
                END_IF;
                IF _retval = WORD#8094 THEN
                    Messenger.Activate(UINT#892,eAxoMessageCategory#Error);
                    Status.Error.Id := UINT#892;
                    RETURN;
                END_IF;
                IF _retval = WORD#8095 THEN
                    Messenger.Activate(UINT#893,eAxoMessageCategory#Error);
                    Status.Error.Id := UINT#893;
                    RETURN;
                END_IF;
                IF _retval = WORD#8096 THEN
                    Messenger.Activate(UINT#894,eAxoMessageCategory#Error);
                    Status.Error.Id := UINT#894;
                    RETURN;
                END_IF;
                IF _retval = WORD#8097 THEN
                    Messenger.Activate(UINT#895,eAxoMessageCategory#Error);
                    Status.Error.Id := UINT#895;
                    RETURN;
                END_IF;
                ReadHardwareIOAddress(hardwareID := (Config.HWIDs.HwID_ToolResult_13) , inputStartAddress => _inputsAddress , inputCount => _inputsCount , outputStartAddress => _outputsAddress , outputCount => _outputsCount);
                IF _inputsCount <> UINT#20 OR _outputsCount <> UINT#0 THEN
                    Messenger.Activate(UINT#896,eAxoMessageCategory#Error);
                    Status.Error.Id := UINT#896;
                    RETURN;
                END_IF;
                //******************Slot 20*****************//
                _geoAddr.Slot   :=  UINT#20;
                _geoAddr.HardwareType := UINT#4; // (4-Module)
                _retval := ReadHardwareIDFromSlot(geoAddr := _geoAddr, hardwareID => Config.HWIDs.HwID_ToolResult_14);
                IF Config.HWIDs.HwID_ToolResult_14 = UINT#0 THEN
                    Messenger.Activate(UINT#900,eAxoMessageCategory#Error);
                    Status.Error.Id := UINT#900;
                    RETURN;
                END_IF;
                IF _retval = WORD#8091 THEN
                    Messenger.Activate(UINT#901,eAxoMessageCategory#Error);
                    Status.Error.Id := UINT#901;
                    RETURN;
                END_IF;
                IF _retval = WORD#8094 THEN
                    Messenger.Activate(UINT#902,eAxoMessageCategory#Error);
                    Status.Error.Id := UINT#902;
                    RETURN;
                END_IF;
                IF _retval = WORD#8095 THEN
                    Messenger.Activate(UINT#903,eAxoMessageCategory#Error);
                    Status.Error.Id := UINT#903;
                    RETURN;
                END_IF;
                IF _retval = WORD#8096 THEN
                    Messenger.Activate(UINT#904,eAxoMessageCategory#Error);
                    Status.Error.Id := UINT#904;
                    RETURN;
                END_IF;
                IF _retval = WORD#8097 THEN
                    Messenger.Activate(UINT#905,eAxoMessageCategory#Error);
                    Status.Error.Id := UINT#905;
                    RETURN;
                END_IF;
                ReadHardwareIOAddress(hardwareID := (Config.HWIDs.HwID_ToolResult_14) , inputStartAddress => _inputsAddress , inputCount => _inputsCount , outputStartAddress => _outputsAddress , outputCount => _outputsCount);
                IF _inputsCount <> UINT#20 OR _outputsCount <> UINT#0 THEN
                    Messenger.Activate(UINT#916,eAxoMessageCategory#Error);
                    Status.Error.Id := UINT#916;
                    RETURN;
                END_IF;
                //******************Slot 21*****************//
                _geoAddr.Slot   :=  UINT#21;
                _geoAddr.HardwareType := UINT#4; // (4-Module)
                _retval := ReadHardwareIDFromSlot(geoAddr := _geoAddr, hardwareID => Config.HWIDs.HwID_ToolResult_15);
                IF Config.HWIDs.HwID_ToolResult_15 = UINT#0 THEN
                    Messenger.Activate(UINT#910,eAxoMessageCategory#Error);
                    Status.Error.Id := UINT#910;
                    RETURN;
                END_IF;
                IF _retval = WORD#8091 THEN
                    Messenger.Activate(UINT#911,eAxoMessageCategory#Error);
                    Status.Error.Id := UINT#911;
                    RETURN;
                END_IF;
                IF _retval = WORD#8094 THEN
                    Messenger.Activate(UINT#912,eAxoMessageCategory#Error);
                    Status.Error.Id := UINT#912;
                    RETURN;
                END_IF;
                IF _retval = WORD#8095 THEN
                    Messenger.Activate(UINT#913,eAxoMessageCategory#Error);
                    Status.Error.Id := UINT#913;
                    RETURN;
                END_IF;
                IF _retval = WORD#8096 THEN
                    Messenger.Activate(UINT#914,eAxoMessageCategory#Error);
                    Status.Error.Id := UINT#914;
                    RETURN;
                END_IF;
                IF _retval = WORD#8097 THEN
                    Messenger.Activate(UINT#715,eAxoMessageCategory#Error);
                    Status.Error.Id := UINT#715;
                    RETURN;
                END_IF;
                ReadHardwareIOAddress(hardwareID := (Config.HWIDs.HwID_ToolResult_15) , inputStartAddress => _inputsAddress , inputCount => _inputsCount , outputStartAddress => _outputsAddress , outputCount => _outputsCount);
                IF _inputsCount <> UINT#20 OR _outputsCount <> UINT#0 THEN
                    Messenger.Activate(UINT#916,eAxoMessageCategory#Error);
                    Status.Error.Id := UINT#916;
                    RETURN;
                END_IF;
                //******************Slot 22*****************//
                _geoAddr.Slot   :=  UINT#22;
                _geoAddr.HardwareType := UINT#4; // (4-Module)
                _retval := ReadHardwareIDFromSlot(geoAddr := _geoAddr, hardwareID => Config.HWIDs.HwID_ToolResult_16);
                IF Config.HWIDs.HwID_ToolResult_16 = UINT#0 THEN
                    Messenger.Activate(UINT#920,eAxoMessageCategory#Error);
                    Status.Error.Id := UINT#920;
                    RETURN;
                END_IF;
                IF _retval = WORD#8091 THEN
                    Messenger.Activate(UINT#921,eAxoMessageCategory#Error);
                    Status.Error.Id := UINT#921;
                    RETURN;
                END_IF;
                IF _retval = WORD#8094 THEN
                    Messenger.Activate(UINT#922,eAxoMessageCategory#Error);
                    Status.Error.Id := UINT#922;
                    RETURN;
                END_IF;
                IF _retval = WORD#8095 THEN
                    Messenger.Activate(UINT#923,eAxoMessageCategory#Error);
                    Status.Error.Id := UINT#923;
                    RETURN;
                END_IF;
                IF _retval = WORD#8096 THEN
                    Messenger.Activate(UINT#924,eAxoMessageCategory#Error);
                    Status.Error.Id := UINT#924;
                    RETURN;
                END_IF;
                IF _retval = WORD#8097 THEN
                    Messenger.Activate(UINT#925,eAxoMessageCategory#Error);
                    Status.Error.Id := UINT#925;
                    RETURN;
                END_IF;
                ReadHardwareIOAddress(hardwareID := (Config.HWIDs.HwID_ToolResult_16) , inputStartAddress => _inputsAddress , inputCount => _inputsCount , outputStartAddress => _outputsAddress , outputCount => _outputsCount);
                IF _inputsCount <> UINT#20 OR _outputsCount <> UINT#0 THEN
                    Messenger.Activate(UINT#926,eAxoMessageCategory#Error);
                    Status.Error.Id := UINT#926;
                    RETURN;
                END_IF;
                //******************Slot 23*****************//
                _geoAddr.Slot   :=  UINT#23;
                _geoAddr.HardwareType := UINT#4; // (4-Module)
                _retval := ReadHardwareIDFromSlot(geoAddr := _geoAddr, hardwareID => Config.HWIDs.HwID_ToolResult_17);
                IF Config.HWIDs.HwID_ToolResult_17 = UINT#0 THEN
                    Messenger.Activate(UINT#930,eAxoMessageCategory#Error);
                    Status.Error.Id := UINT#930;
                    RETURN;
                END_IF;
                IF _retval = WORD#8091 THEN
                    Messenger.Activate(UINT#931,eAxoMessageCategory#Error);
                    Status.Error.Id := UINT#931;
                    RETURN;
                END_IF;
                IF _retval = WORD#8094 THEN
                    Messenger.Activate(UINT#932,eAxoMessageCategory#Error);
                    Status.Error.Id := UINT#932;
                    RETURN;
                END_IF;
                IF _retval = WORD#8095 THEN
                    Messenger.Activate(UINT#933,eAxoMessageCategory#Error);
                    Status.Error.Id := UINT#933;
                    RETURN;
                END_IF;
                IF _retval = WORD#8096 THEN
                    Messenger.Activate(UINT#934,eAxoMessageCategory#Error);
                    Status.Error.Id := UINT#934;
                    RETURN;
                END_IF;
                IF _retval = WORD#8097 THEN
                    Messenger.Activate(UINT#935,eAxoMessageCategory#Error);
                    Status.Error.Id := UINT#935;
                    RETURN;
                END_IF;
                ReadHardwareIOAddress(hardwareID := (Config.HWIDs.HwID_ToolResult_17) , inputStartAddress => _inputsAddress , inputCount => _inputsCount , outputStartAddress => _outputsAddress , outputCount => _outputsCount);
                IF _inputsCount <> UINT#20 OR _outputsCount <> UINT#0 THEN
                    Messenger.Activate(UINT#936,eAxoMessageCategory#Error);
                    Status.Error.Id := UINT#936;
                    RETURN;
                END_IF;
                //******************Slot 24*****************//
                _geoAddr.Slot   :=  UINT#24;
                _geoAddr.HardwareType := UINT#4; // (4-Module)
                _retval := ReadHardwareIDFromSlot(geoAddr := _geoAddr, hardwareID => Config.HWIDs.HwID_ToolResult_18);
                IF Config.HWIDs.HwID_ToolResult_18 = UINT#0 THEN
                    Messenger.Activate(UINT#940,eAxoMessageCategory#Error);
                    Status.Error.Id := UINT#940;
                    RETURN;
                END_IF;
                IF _retval = WORD#8091 THEN
                    Messenger.Activate(UINT#941,eAxoMessageCategory#Error);
                    Status.Error.Id := UINT#941;
                    RETURN;
                END_IF;
                IF _retval = WORD#8094 THEN
                    Messenger.Activate(UINT#942,eAxoMessageCategory#Error);
                    Status.Error.Id := UINT#942;
                    RETURN;
                END_IF;
                IF _retval = WORD#8095 THEN
                    Messenger.Activate(UINT#943,eAxoMessageCategory#Error);
                    Status.Error.Id := UINT#943;
                    RETURN;
                END_IF;
                IF _retval = WORD#8096 THEN
                    Messenger.Activate(UINT#944,eAxoMessageCategory#Error);
                    Status.Error.Id := UINT#944;
                    RETURN;
                END_IF;
                IF _retval = WORD#8097 THEN
                    Messenger.Activate(UINT#945,eAxoMessageCategory#Error);
                    Status.Error.Id := UINT#945;
                    RETURN;
                END_IF;
                ReadHardwareIOAddress(hardwareID := (Config.HWIDs.HwID_ToolResult_18) , inputStartAddress => _inputsAddress , inputCount => _inputsCount , outputStartAddress => _outputsAddress , outputCount => _outputsCount);
                IF _inputsCount <> UINT#20 OR _outputsCount <> UINT#0 THEN
                    Messenger.Activate(UINT#946,eAxoMessageCategory#Error);
                    Status.Error.Id := UINT#946;
                    RETURN;
                END_IF;
                //******************Slot 25*****************//
                _geoAddr.Slot   :=  UINT#25;
                _geoAddr.HardwareType := UINT#4; // (4-Module)
                _retval := ReadHardwareIDFromSlot(geoAddr := _geoAddr, hardwareID => Config.HWIDs.HwID_ToolResult_19);
                IF Config.HWIDs.HwID_ToolResult_19 = UINT#0 THEN
                    Messenger.Activate(UINT#950,eAxoMessageCategory#Error);
                    Status.Error.Id := UINT#950;
                    RETURN;
                END_IF;
                IF _retval = WORD#8091 THEN
                    Messenger.Activate(UINT#951,eAxoMessageCategory#Error);
                    Status.Error.Id := UINT#951;
                    RETURN;
                END_IF;
                IF _retval = WORD#8094 THEN
                    Messenger.Activate(UINT#952,eAxoMessageCategory#Error);
                    Status.Error.Id := UINT#952;
                    RETURN;
                END_IF;
                IF _retval = WORD#8095 THEN
                    Messenger.Activate(UINT#953,eAxoMessageCategory#Error);
                    Status.Error.Id := UINT#953;
                    RETURN;
                END_IF;
                IF _retval = WORD#8096 THEN
                    Messenger.Activate(UINT#954,eAxoMessageCategory#Error);
                    Status.Error.Id := UINT#954;
                    RETURN;
                END_IF;
                IF _retval = WORD#8097 THEN
                    Messenger.Activate(UINT#955,eAxoMessageCategory#Error);
                    Status.Error.Id := UINT#955;
                    RETURN;
                END_IF;
                ReadHardwareIOAddress(hardwareID := (Config.HWIDs.HwID_ToolResult_19) , inputStartAddress => _inputsAddress , inputCount => _inputsCount , outputStartAddress => _outputsAddress , outputCount => _outputsCount);
                IF _inputsCount <> UINT#20 OR _outputsCount <> UINT#0 THEN
                    Messenger.Activate(UINT#956,eAxoMessageCategory#Error);
                    Status.Error.Id := UINT#956;
                    RETURN;
                END_IF;
                //******************Slot 26*****************//
                _geoAddr.Slot   :=  UINT#26;
                _geoAddr.HardwareType := UINT#4; // (4-Module)
                _retval := ReadHardwareIDFromSlot(geoAddr := _geoAddr, hardwareID => Config.HWIDs.HwID_ToolResult_20);
                IF Config.HWIDs.HwID_ToolResult_20 = UINT#0 THEN
                    Messenger.Activate(UINT#960,eAxoMessageCategory#Error);
                    Status.Error.Id := UINT#960;
                    RETURN;
                END_IF;
                IF _retval = WORD#8091 THEN
                    Messenger.Activate(UINT#961,eAxoMessageCategory#Error);
                    Status.Error.Id := UINT#961;
                    RETURN;
                END_IF;
                IF _retval = WORD#8094 THEN
                    Messenger.Activate(UINT#962,eAxoMessageCategory#Error);
                    Status.Error.Id := UINT#962;
                    RETURN;
                END_IF;
                IF _retval = WORD#8095 THEN
                    Messenger.Activate(UINT#963,eAxoMessageCategory#Error);
                    Status.Error.Id := UINT#963;
                    RETURN;
                END_IF;
                IF _retval = WORD#8096 THEN
                    Messenger.Activate(UINT#964,eAxoMessageCategory#Error);
                    Status.Error.Id := UINT#964;
                    RETURN;
                END_IF;
                IF _retval = WORD#8097 THEN
                    Messenger.Activate(UINT#965,eAxoMessageCategory#Error);
                    Status.Error.Id := UINT#965;
                    RETURN;
                END_IF;
                ReadHardwareIOAddress(hardwareID := (Config.HWIDs.HwID_ToolResult_20) , inputStartAddress => _inputsAddress , inputCount => _inputsCount , outputStartAddress => _outputsAddress , outputCount => _outputsCount);
                IF _inputsCount <> UINT#20 OR _outputsCount <> UINT#0 THEN
                    Messenger.Activate(UINT#966,eAxoMessageCategory#Error);
                    Status.Error.Id := UINT#966;
                    RETURN;
                END_IF;
                //******************Slot 27*****************//
                _geoAddr.Slot   :=  UINT#27;
                _geoAddr.HardwareType := UINT#4; // (4-Module)
                _retval := ReadHardwareIDFromSlot(geoAddr := _geoAddr, hardwareID => Config.HWIDs.HwID_ToolResult_21);
                IF Config.HWIDs.HwID_ToolResult_21 = UINT#0 THEN
                    Messenger.Activate(UINT#970,eAxoMessageCategory#Error);
                    Status.Error.Id := UINT#970;
                    RETURN;
                END_IF;
                IF _retval = WORD#8091 THEN
                    Messenger.Activate(UINT#971,eAxoMessageCategory#Error);
                    Status.Error.Id := UINT#971;
                    RETURN;
                END_IF;
                IF _retval = WORD#8094 THEN
                    Messenger.Activate(UINT#972,eAxoMessageCategory#Error);
                    Status.Error.Id := UINT#972;
                    RETURN;
                END_IF;
                IF _retval = WORD#8095 THEN
                    Messenger.Activate(UINT#973,eAxoMessageCategory#Error);
                    Status.Error.Id := UINT#973;
                    RETURN;
                END_IF;
                IF _retval = WORD#8096 THEN
                    Messenger.Activate(UINT#974,eAxoMessageCategory#Error);
                    Status.Error.Id := UINT#974;
                    RETURN;
                END_IF;
                IF _retval = WORD#8097 THEN
                    Messenger.Activate(UINT#975,eAxoMessageCategory#Error);
                    Status.Error.Id := UINT#975;
                    RETURN;
                END_IF;
                ReadHardwareIOAddress(hardwareID := (Config.HWIDs.HwID_ToolResult_21) , inputStartAddress => _inputsAddress , inputCount => _inputsCount , outputStartAddress => _outputsAddress , outputCount => _outputsCount);
                IF _inputsCount <> UINT#20 OR _outputsCount <> UINT#0 THEN
                    Messenger.Activate(UINT#976,eAxoMessageCategory#Error);
                    Status.Error.Id := UINT#976;
                    RETURN;
                END_IF;
                //******************Slot 28*****************//
                _geoAddr.Slot   :=  UINT#28;
                _geoAddr.HardwareType := UINT#4; // (4-Module)
                _retval := ReadHardwareIDFromSlot(geoAddr := _geoAddr, hardwareID => Config.HWIDs.HwID_ToolResult_22);
                IF Config.HWIDs.HwID_ToolResult_22 = UINT#0 THEN
                    Messenger.Activate(UINT#980,eAxoMessageCategory#Error);
                    Status.Error.Id := UINT#980;
                    RETURN;
                END_IF;
                IF _retval = WORD#8091 THEN
                    Messenger.Activate(UINT#981,eAxoMessageCategory#Error);
                    Status.Error.Id := UINT#981;
                    RETURN;
                END_IF;
                IF _retval = WORD#8094 THEN
                    Messenger.Activate(UINT#982,eAxoMessageCategory#Error);
                    Status.Error.Id := UINT#982;
                    RETURN;
                END_IF;
                IF _retval = WORD#8095 THEN
                    Messenger.Activate(UINT#983,eAxoMessageCategory#Error);
                    Status.Error.Id := UINT#983;
                    RETURN;
                END_IF;
                IF _retval = WORD#8096 THEN
                    Messenger.Activate(UINT#984,eAxoMessageCategory#Error);
                    Status.Error.Id := UINT#984;
                    RETURN;
                END_IF;
                IF _retval = WORD#8097 THEN
                    Messenger.Activate(UINT#985,eAxoMessageCategory#Error);
                    Status.Error.Id := UINT#985;
                    RETURN;
                END_IF;
                ReadHardwareIOAddress(hardwareID := (Config.HWIDs.HwID_ToolResult_22) , inputStartAddress => _inputsAddress , inputCount => _inputsCount , outputStartAddress => _outputsAddress , outputCount => _outputsCount);
                IF _inputsCount <> UINT#20 OR _outputsCount <> UINT#0 THEN
                    Messenger.Activate(UINT#986,eAxoMessageCategory#Error);
                    Status.Error.Id := UINT#986;
                    RETURN;
                END_IF;
                //******************Slot 29*****************//
                _geoAddr.Slot   :=  UINT#29;
                _geoAddr.HardwareType := UINT#4; // (4-Module)
                _retval := ReadHardwareIDFromSlot(geoAddr := _geoAddr, hardwareID => Config.HWIDs.HwID_ToolResult_23);
                IF Config.HWIDs.HwID_ToolResult_23 = UINT#0 THEN
                    Messenger.Activate(UINT#990,eAxoMessageCategory#Error);
                    Status.Error.Id := UINT#990;
                    RETURN;
                END_IF;
                IF _retval = WORD#8091 THEN
                    Messenger.Activate(UINT#991,eAxoMessageCategory#Error);
                    Status.Error.Id := UINT#991;
                    RETURN;
                END_IF;
                IF _retval = WORD#8094 THEN
                    Messenger.Activate(UINT#992,eAxoMessageCategory#Error);
                    Status.Error.Id := UINT#992;
                    RETURN;
                END_IF;
                IF _retval = WORD#8095 THEN
                    Messenger.Activate(UINT#993,eAxoMessageCategory#Error);
                    Status.Error.Id := UINT#993;
                    RETURN;
                END_IF;
                IF _retval = WORD#8096 THEN
                    Messenger.Activate(UINT#994,eAxoMessageCategory#Error);
                    Status.Error.Id := UINT#994;
                    RETURN;
                END_IF;
                IF _retval = WORD#8097 THEN
                    Messenger.Activate(UINT#995,eAxoMessageCategory#Error);
                    Status.Error.Id := UINT#995;
                    RETURN;
                END_IF;
                ReadHardwareIOAddress(hardwareID := (Config.HWIDs.HwID_ToolResult_23) , inputStartAddress => _inputsAddress , inputCount => _inputsCount , outputStartAddress => _outputsAddress , outputCount => _outputsCount);
                IF _inputsCount <> UINT#20 OR _outputsCount <> UINT#0 THEN
                    Messenger.Activate(UINT#996,eAxoMessageCategory#Error);
                    Status.Error.Id := UINT#996;
                    RETURN;
                END_IF;
                //******************Slot 30*****************//
                _geoAddr.Slot   :=  UINT#30;
                _geoAddr.HardwareType := UINT#4; // (4-Module)
                _retval := ReadHardwareIDFromSlot(geoAddr := _geoAddr, hardwareID => Config.HWIDs.HwID_ToolResult_24);
                IF Config.HWIDs.HwID_ToolResult_24 = UINT#0 THEN
                    Messenger.Activate(UINT#1000,eAxoMessageCategory#Error);
                    Status.Error.Id := UINT#1000;
                    RETURN;
                END_IF;
                IF _retval = WORD#8091 THEN
                    Messenger.Activate(UINT#1001,eAxoMessageCategory#Error);
                    Status.Error.Id := UINT#1001;
                    RETURN;
                END_IF;
                IF _retval = WORD#8094 THEN
                    Messenger.Activate(UINT#1002,eAxoMessageCategory#Error);
                    Status.Error.Id := UINT#1002;
                    RETURN;
                END_IF;
                IF _retval = WORD#8095 THEN
                    Messenger.Activate(UINT#1003,eAxoMessageCategory#Error);
                    Status.Error.Id := UINT#1003;
                    RETURN;
                END_IF;
                IF _retval = WORD#8096 THEN
                    Messenger.Activate(UINT#1004,eAxoMessageCategory#Error);
                    Status.Error.Id := UINT#1004;
                    RETURN;
                END_IF;
                IF _retval = WORD#8097 THEN
                    Messenger.Activate(UINT#1005,eAxoMessageCategory#Error);
                    Status.Error.Id := UINT#1005;
                    RETURN;
                END_IF;
                ReadHardwareIOAddress(hardwareID := (Config.HWIDs.HwID_ToolResult_24) , inputStartAddress => _inputsAddress , inputCount => _inputsCount , outputStartAddress => _outputsAddress , outputCount => _outputsCount);
                IF _inputsCount <> UINT#20 OR _outputsCount <> UINT#0 THEN
                    Messenger.Activate(UINT#1006,eAxoMessageCategory#Error);
                    Status.Error.Id := UINT#1006;
                    RETURN;
                END_IF;
                //******************Slot 31*****************//
                _geoAddr.Slot   :=  UINT#31;
                _geoAddr.HardwareType := UINT#4; // (4-Module)
                _retval := ReadHardwareIDFromSlot(geoAddr := _geoAddr, hardwareID => Config.HWIDs.HwID_ToolResult_25);
                IF Config.HWIDs.HwID_ToolResult_25 = UINT#0 THEN
                    Messenger.Activate(UINT#1010,eAxoMessageCategory#Error);
                    Status.Error.Id := UINT#1010;
                    RETURN;
                END_IF;
                IF _retval = WORD#8091 THEN
                    Messenger.Activate(UINT#1011,eAxoMessageCategory#Error);
                    Status.Error.Id := UINT#1011;
                    RETURN;
                END_IF;
                IF _retval = WORD#8094 THEN
                    Messenger.Activate(UINT#1012,eAxoMessageCategory#Error);
                    Status.Error.Id := UINT#1012;
                    RETURN;
                END_IF;
                IF _retval = WORD#8095 THEN
                    Messenger.Activate(UINT#1013,eAxoMessageCategory#Error);
                    Status.Error.Id := UINT#1013;
                    RETURN;
                END_IF;
                IF _retval = WORD#8096 THEN
                    Messenger.Activate(UINT#1014,eAxoMessageCategory#Error);
                    Status.Error.Id := UINT#1014;
                    RETURN;
                END_IF;
                IF _retval = WORD#8097 THEN
                    Messenger.Activate(UINT#1015,eAxoMessageCategory#Error);
                    Status.Error.Id := UINT#1015;
                    RETURN;
                END_IF;
                ReadHardwareIOAddress(hardwareID := (Config.HWIDs.HwID_ToolResult_25) , inputStartAddress => _inputsAddress , inputCount => _inputsCount , outputStartAddress => _outputsAddress , outputCount => _outputsCount);
                IF _inputsCount <> UINT#20 OR _outputsCount <> UINT#0 THEN
                    Messenger.Activate(UINT#1016,eAxoMessageCategory#Error);
                    Status.Error.Id := UINT#1016;
                    RETURN;
                END_IF;
                //******************Slot 32*****************//
                _geoAddr.Slot   :=  UINT#32;
                _geoAddr.HardwareType := UINT#4; // (4-Module)
                _retval := ReadHardwareIDFromSlot(geoAddr := _geoAddr, hardwareID => Config.HWIDs.HwID_ToolResult_26);
                IF Config.HWIDs.HwID_ToolResult_26 = UINT#0 THEN
                    Messenger.Activate(UINT#1020,eAxoMessageCategory#Error);
                    Status.Error.Id := UINT#1020;
                    RETURN;
                END_IF;
                IF _retval = WORD#8091 THEN
                    Messenger.Activate(UINT#1021,eAxoMessageCategory#Error);
                    Status.Error.Id := UINT#1021;
                    RETURN;
                END_IF;
                IF _retval = WORD#8094 THEN
                    Messenger.Activate(UINT#1022,eAxoMessageCategory#Error);
                    Status.Error.Id := UINT#1022;
                    RETURN;
                END_IF;
                IF _retval = WORD#8095 THEN
                    Messenger.Activate(UINT#1023,eAxoMessageCategory#Error);
                    Status.Error.Id := UINT#1023;
                    RETURN;
                END_IF;
                IF _retval = WORD#8096 THEN
                    Messenger.Activate(UINT#1024,eAxoMessageCategory#Error);
                    Status.Error.Id := UINT#1024;
                    RETURN;
                END_IF;
                IF _retval = WORD#8097 THEN
                    Messenger.Activate(UINT#1025,eAxoMessageCategory#Error);
                    Status.Error.Id := UINT#1025;
                    RETURN;
                END_IF;
                ReadHardwareIOAddress(hardwareID := (Config.HWIDs.HwID_ToolResult_26) , inputStartAddress => _inputsAddress , inputCount => _inputsCount , outputStartAddress => _outputsAddress , outputCount => _outputsCount);
                IF _inputsCount <> UINT#20 OR _outputsCount <> UINT#0 THEN
                    Messenger.Activate(UINT#1026,eAxoMessageCategory#Error);
                    Status.Error.Id := UINT#1026;
                    RETURN;
                END_IF;
                //******************Slot 33*****************//
                _geoAddr.Slot   :=  UINT#33;
                _geoAddr.HardwareType := UINT#4; // (4-Module)
                _retval := ReadHardwareIDFromSlot(geoAddr := _geoAddr, hardwareID => Config.HWIDs.HwID_ToolResult_27);
                IF Config.HWIDs.HwID_ToolResult_27 = UINT#0 THEN
                    Messenger.Activate(UINT#1030,eAxoMessageCategory#Error);
                    Status.Error.Id := UINT#1030;
                    RETURN;
                END_IF;
                IF _retval = WORD#8091 THEN
                    Messenger.Activate(UINT#1031,eAxoMessageCategory#Error);
                    Status.Error.Id := UINT#1031;
                    RETURN;
                END_IF;
                IF _retval = WORD#8094 THEN
                    Messenger.Activate(UINT#1032,eAxoMessageCategory#Error);
                    Status.Error.Id := UINT#1032;
                    RETURN;
                END_IF;
                IF _retval = WORD#8095 THEN
                    Messenger.Activate(UINT#1033,eAxoMessageCategory#Error);
                    Status.Error.Id := UINT#1033;
                    RETURN;
                END_IF;
                IF _retval = WORD#8096 THEN
                    Messenger.Activate(UINT#1034,eAxoMessageCategory#Error);
                    Status.Error.Id := UINT#1034;
                    RETURN;
                END_IF;
                IF _retval = WORD#8097 THEN
                    Messenger.Activate(UINT#1035,eAxoMessageCategory#Error);
                    Status.Error.Id := UINT#1035;
                    RETURN;
                END_IF;
                ReadHardwareIOAddress(hardwareID := (Config.HWIDs.HwID_ToolResult_27) , inputStartAddress => _inputsAddress , inputCount => _inputsCount , outputStartAddress => _outputsAddress , outputCount => _outputsCount);
                IF _inputsCount <> UINT#20 OR _outputsCount <> UINT#0 THEN
                    Messenger.Activate(UINT#1036,eAxoMessageCategory#Error);
                    Status.Error.Id := UINT#1036;
                    RETURN;
                END_IF;
                //******************Slot 34*****************//
                _geoAddr.Slot   :=  UINT#34;
                _geoAddr.HardwareType := UINT#4; // (4-Module)
                _retval := ReadHardwareIDFromSlot(geoAddr := _geoAddr, hardwareID => Config.HWIDs.HwID_ToolResult_28);
                IF Config.HWIDs.HwID_ToolResult_28 = UINT#0 THEN
                    Messenger.Activate(UINT#1040,eAxoMessageCategory#Error);
                    Status.Error.Id := UINT#1040;
                    RETURN;
                END_IF;
                IF _retval = WORD#8091 THEN
                    Messenger.Activate(UINT#1041,eAxoMessageCategory#Error);
                    Status.Error.Id := UINT#1041;
                    RETURN;
                END_IF;
                IF _retval = WORD#8094 THEN
                    Messenger.Activate(UINT#1042,eAxoMessageCategory#Error);
                    Status.Error.Id := UINT#1042;
                    RETURN;
                END_IF;
                IF _retval = WORD#8095 THEN
                    Messenger.Activate(UINT#1043,eAxoMessageCategory#Error);
                    Status.Error.Id := UINT#1043;
                    RETURN;
                END_IF;
                IF _retval = WORD#8096 THEN
                    Messenger.Activate(UINT#1044,eAxoMessageCategory#Error);
                    Status.Error.Id := UINT#1044;
                    RETURN;
                END_IF;
                IF _retval = WORD#8097 THEN
                    Messenger.Activate(UINT#1045,eAxoMessageCategory#Error);
                    Status.Error.Id := UINT#1045;
                    RETURN;
                END_IF;
                ReadHardwareIOAddress(hardwareID := (Config.HWIDs.HwID_ToolResult_28) , inputStartAddress => _inputsAddress , inputCount => _inputsCount , outputStartAddress => _outputsAddress , outputCount => _outputsCount);
                IF _inputsCount <> UINT#20 OR _outputsCount <> UINT#0 THEN
                    Messenger.Activate(UINT#1046,eAxoMessageCategory#Error);
                    Status.Error.Id := UINT#1046;
                    RETURN;
                END_IF;
                //******************Slot 35*****************//
                _geoAddr.Slot   :=  UINT#35;
                _geoAddr.HardwareType := UINT#4; // (4-Module)
                _retval := ReadHardwareIDFromSlot(geoAddr := _geoAddr, hardwareID => Config.HWIDs.HwID_ToolResult_29);
                IF Config.HWIDs.HwID_ToolResult_29 = UINT#0 THEN
                    Messenger.Activate(UINT#1050,eAxoMessageCategory#Error);
                    Status.Error.Id := UINT#1050;
                    RETURN;
                END_IF;
                IF _retval = WORD#8091 THEN
                    Messenger.Activate(UINT#1051,eAxoMessageCategory#Error);
                    Status.Error.Id := UINT#1051;
                    RETURN;
                END_IF;
                IF _retval = WORD#8094 THEN
                    Messenger.Activate(UINT#1052,eAxoMessageCategory#Error);
                    Status.Error.Id := UINT#1052;
                    RETURN;
                END_IF;
                IF _retval = WORD#8095 THEN
                    Messenger.Activate(UINT#1053,eAxoMessageCategory#Error);
                    Status.Error.Id := UINT#1053;
                    RETURN;
                END_IF;
                IF _retval = WORD#8096 THEN
                    Messenger.Activate(UINT#1054,eAxoMessageCategory#Error);
                    Status.Error.Id := UINT#1054;
                    RETURN;
                END_IF;
                IF _retval = WORD#8097 THEN
                    Messenger.Activate(UINT#1055,eAxoMessageCategory#Error);
                    Status.Error.Id := UINT#1055;
                    RETURN;
                END_IF;
                ReadHardwareIOAddress(hardwareID := (Config.HWIDs.HwID_ToolResult_29) , inputStartAddress => _inputsAddress , inputCount => _inputsCount , outputStartAddress => _outputsAddress , outputCount => _outputsCount);
                IF _inputsCount <> UINT#20 OR _outputsCount <> UINT#0 THEN
                    Messenger.Activate(UINT#1056,eAxoMessageCategory#Error);
                    Status.Error.Id := UINT#1056;
                    RETURN;
                END_IF;
                //******************Slot 36*****************//
                _geoAddr.Slot   :=  UINT#36;
                _geoAddr.HardwareType := UINT#4; // (4-Module)
                _retval := ReadHardwareIDFromSlot(geoAddr := _geoAddr, hardwareID => Config.HWIDs.HwID_ToolResult_30);
                IF Config.HWIDs.HwID_ToolResult_30 = UINT#0 THEN
                    Messenger.Activate(UINT#1060,eAxoMessageCategory#Error);
                    Status.Error.Id := UINT#1060;
                    RETURN;
                END_IF;
                IF _retval = WORD#8091 THEN
                    Messenger.Activate(UINT#1061,eAxoMessageCategory#Error);
                    Status.Error.Id := UINT#1061;
                    RETURN;
                END_IF;
                IF _retval = WORD#8094 THEN
                    Messenger.Activate(UINT#1062,eAxoMessageCategory#Error);
                    Status.Error.Id := UINT#1062;
                    RETURN;
                END_IF;
                IF _retval = WORD#8095 THEN
                    Messenger.Activate(UINT#1063,eAxoMessageCategory#Error);
                    Status.Error.Id := UINT#1063;
                    RETURN;
                END_IF;
                IF _retval = WORD#8096 THEN
                    Messenger.Activate(UINT#1064,eAxoMessageCategory#Error);
                    Status.Error.Id := UINT#1064;
                    RETURN;
                END_IF;
                IF _retval = WORD#8097 THEN
                    Messenger.Activate(UINT#1065,eAxoMessageCategory#Error);
                    Status.Error.Id := UINT#1065;
                    RETURN;
                END_IF;
                ReadHardwareIOAddress(hardwareID := (Config.HWIDs.HwID_ToolResult_30) , inputStartAddress => _inputsAddress , inputCount => _inputsCount , outputStartAddress => _outputsAddress , outputCount => _outputsCount);
                IF _inputsCount <> UINT#20 OR _outputsCount <> UINT#0 THEN
                    Messenger.Activate(UINT#1066,eAxoMessageCategory#Error);
                    Status.Error.Id := UINT#1066;
                    RETURN;
                END_IF;
                //******************Slot 37*****************//
                _geoAddr.Slot   :=  UINT#37;
                _geoAddr.HardwareType := UINT#4; // (4-Module)
                _retval := ReadHardwareIDFromSlot(geoAddr := _geoAddr, hardwareID => Config.HWIDs.HwID_ToolResult_31);
                IF Config.HWIDs.HwID_ToolResult_31 = UINT#0 THEN
                    Messenger.Activate(UINT#1070,eAxoMessageCategory#Error);
                    Status.Error.Id := UINT#1070;
                    RETURN;
                END_IF;
                IF _retval = WORD#8091 THEN
                    Messenger.Activate(UINT#1071,eAxoMessageCategory#Error);
                    Status.Error.Id := UINT#1071;
                    RETURN;
                END_IF;
                IF _retval = WORD#8094 THEN
                    Messenger.Activate(UINT#1072,eAxoMessageCategory#Error);
                    Status.Error.Id := UINT#1072;
                    RETURN;
                END_IF;
                IF _retval = WORD#8095 THEN
                    Messenger.Activate(UINT#1073,eAxoMessageCategory#Error);
                    Status.Error.Id := UINT#1073;
                    RETURN;
                END_IF;
                IF _retval = WORD#8096 THEN
                    Messenger.Activate(UINT#1074,eAxoMessageCategory#Error);
                    Status.Error.Id := UINT#1074;
                    RETURN;
                END_IF;
                IF _retval = WORD#8097 THEN
                    Messenger.Activate(UINT#1075,eAxoMessageCategory#Error);
                    Status.Error.Id := UINT#1075;
                    RETURN;
                END_IF;
                ReadHardwareIOAddress(hardwareID := (Config.HWIDs.HwID_ToolResult_31) , inputStartAddress => _inputsAddress , inputCount => _inputsCount , outputStartAddress => _outputsAddress , outputCount => _outputsCount);
                IF _inputsCount <> UINT#20 OR _outputsCount <> UINT#0 THEN
                    Messenger.Activate(UINT#1076,eAxoMessageCategory#Error);
                    Status.Error.Id := UINT#1076;
                    RETURN;
                END_IF;
                //******************Slot 38*****************//
                _geoAddr.Slot   :=  UINT#38;
                _geoAddr.HardwareType := UINT#4; // (4-Module)
                _retval := ReadHardwareIDFromSlot(geoAddr := _geoAddr, hardwareID => Config.HWIDs.HwID_ToolResult_32);
                IF Config.HWIDs.HwID_ToolResult_32 = UINT#0 THEN
                    Messenger.Activate(UINT#1080,eAxoMessageCategory#Error);
                    Status.Error.Id := UINT#1080;
                    RETURN;
                END_IF;
                IF _retval = WORD#8091 THEN
                    Messenger.Activate(UINT#1081,eAxoMessageCategory#Error);
                    Status.Error.Id := UINT#1081;
                    RETURN;
                END_IF;
                IF _retval = WORD#8094 THEN
                    Messenger.Activate(UINT#1082,eAxoMessageCategory#Error);
                    Status.Error.Id := UINT#1082;
                    RETURN;
                END_IF;
                IF _retval = WORD#8095 THEN
                    Messenger.Activate(UINT#1083,eAxoMessageCategory#Error);
                    Status.Error.Id := UINT#1083;
                    RETURN;
                END_IF;
                IF _retval = WORD#8096 THEN
                    Messenger.Activate(UINT#1084,eAxoMessageCategory#Error);
                    Status.Error.Id := UINT#1084;
                    RETURN;
                END_IF;
                IF _retval = WORD#8097 THEN
                    Messenger.Activate(UINT#1085,eAxoMessageCategory#Error);
                    Status.Error.Id := UINT#1085;
                    RETURN;
                END_IF;
                ReadHardwareIOAddress(hardwareID := (Config.HWIDs.HwID_ToolResult_32) , inputStartAddress => _inputsAddress , inputCount => _inputsCount , outputStartAddress => _outputsAddress , outputCount => _outputsCount);
                IF _inputsCount <> UINT#20 OR _outputsCount <> UINT#0 THEN
                    Messenger.Activate(UINT#1086,eAxoMessageCategory#Error);
                    Status.Error.Id := UINT#1086;
                    RETURN;
                END_IF;
                //******************Slot 39*****************//
                _geoAddr.Slot   :=  UINT#39;
                _geoAddr.HardwareType := UINT#4; // (4-Module)
                _retval := ReadHardwareIDFromSlot(geoAddr := _geoAddr, hardwareID => Config.HWIDs.HwID_ToolResult_33);
                IF Config.HWIDs.HwID_ToolResult_33 = UINT#0 THEN
                    Messenger.Activate(UINT#1090,eAxoMessageCategory#Error);
                    Status.Error.Id := UINT#1090;
                    RETURN;
                END_IF;
                IF _retval = WORD#8091 THEN
                    Messenger.Activate(UINT#1091,eAxoMessageCategory#Error);
                    Status.Error.Id := UINT#1091;
                    RETURN;
                END_IF;
                IF _retval = WORD#8094 THEN
                    Messenger.Activate(UINT#1092,eAxoMessageCategory#Error);
                    Status.Error.Id := UINT#1092;
                    RETURN;
                END_IF;
                IF _retval = WORD#8095 THEN
                    Messenger.Activate(UINT#1093,eAxoMessageCategory#Error);
                    Status.Error.Id := UINT#1093;
                    RETURN;
                END_IF;
                IF _retval = WORD#8096 THEN
                    Messenger.Activate(UINT#1094,eAxoMessageCategory#Error);
                    Status.Error.Id := UINT#1094;
                    RETURN;
                END_IF;
                IF _retval = WORD#8097 THEN
                    Messenger.Activate(UINT#1095,eAxoMessageCategory#Error);
                    Status.Error.Id := UINT#1095;
                    RETURN;
                END_IF;
                ReadHardwareIOAddress(hardwareID := (Config.HWIDs.HwID_ToolResult_33) , inputStartAddress => _inputsAddress , inputCount => _inputsCount , outputStartAddress => _outputsAddress , outputCount => _outputsCount);
                IF _inputsCount <> UINT#20 OR _outputsCount <> UINT#0 THEN
                    Messenger.Activate(UINT#1096,eAxoMessageCategory#Error);
                    Status.Error.Id := UINT#1096;
                    RETURN;
                END_IF;
                //******************Slot 40*****************//
                _geoAddr.Slot   :=  UINT#40;
                _geoAddr.HardwareType := UINT#4; // (4-Module)
                _retval := ReadHardwareIDFromSlot(geoAddr := _geoAddr, hardwareID => Config.HWIDs.HwID_ToolResult_34);
                IF Config.HWIDs.HwID_ToolResult_34 = UINT#0 THEN
                    Messenger.Activate(UINT#1100,eAxoMessageCategory#Error);
                    Status.Error.Id := UINT#1100;
                    RETURN;
                END_IF;
                IF _retval = WORD#8091 THEN
                    Messenger.Activate(UINT#1101,eAxoMessageCategory#Error);
                    Status.Error.Id := UINT#1101;
                    RETURN;
                END_IF;
                IF _retval = WORD#8094 THEN
                    Messenger.Activate(UINT#1102,eAxoMessageCategory#Error);
                    Status.Error.Id := UINT#1102;
                    RETURN;
                END_IF;
                IF _retval = WORD#8095 THEN
                    Messenger.Activate(UINT#1103,eAxoMessageCategory#Error);
                    Status.Error.Id := UINT#1103;
                    RETURN;
                END_IF;
                IF _retval = WORD#8096 THEN
                    Messenger.Activate(UINT#1104,eAxoMessageCategory#Error);
                    Status.Error.Id := UINT#1104;
                    RETURN;
                END_IF;
                IF _retval = WORD#8097 THEN
                    Messenger.Activate(UINT#1105,eAxoMessageCategory#Error);
                    Status.Error.Id := UINT#1105;
                    RETURN;
                END_IF;
                ReadHardwareIOAddress(hardwareID := (Config.HWIDs.HwID_ToolResult_34) , inputStartAddress => _inputsAddress , inputCount => _inputsCount , outputStartAddress => _outputsAddress , outputCount => _outputsCount);
                IF _inputsCount <> UINT#20 OR _outputsCount <> UINT#0 THEN
                    Messenger.Activate(UINT#1106,eAxoMessageCategory#Error);
                    Status.Error.Id := UINT#1106;
                    RETURN;
                END_IF;
                //******************Slot 41*****************//
                _geoAddr.Slot   :=  UINT#41;
                _geoAddr.HardwareType := UINT#4; // (4-Module)
                _retval := ReadHardwareIDFromSlot(geoAddr := _geoAddr, hardwareID => Config.HWIDs.HwID_ToolResult_35);
                IF Config.HWIDs.HwID_ToolResult_35 = UINT#0 THEN
                    Messenger.Activate(UINT#1110,eAxoMessageCategory#Error);
                    Status.Error.Id := UINT#1110;
                    RETURN;
                END_IF;
                IF _retval = WORD#8091 THEN
                    Messenger.Activate(UINT#1111,eAxoMessageCategory#Error);
                    Status.Error.Id := UINT#1111;
                    RETURN;
                END_IF;
                IF _retval = WORD#8094 THEN
                    Messenger.Activate(UINT#1112,eAxoMessageCategory#Error);
                    Status.Error.Id := UINT#1112;
                    RETURN;
                END_IF;
                IF _retval = WORD#8095 THEN
                    Messenger.Activate(UINT#1113,eAxoMessageCategory#Error);
                    Status.Error.Id := UINT#1113;
                    RETURN;
                END_IF;
                IF _retval = WORD#8096 THEN
                    Messenger.Activate(UINT#1114,eAxoMessageCategory#Error);
                    Status.Error.Id := UINT#1114;
                    RETURN;
                END_IF;
                IF _retval = WORD#8097 THEN
                    Messenger.Activate(UINT#1115,eAxoMessageCategory#Error);
                    Status.Error.Id := UINT#1115;
                    RETURN;
                END_IF;
                ReadHardwareIOAddress(hardwareID := (Config.HWIDs.HwID_ToolResult_35) , inputStartAddress => _inputsAddress , inputCount => _inputsCount , outputStartAddress => _outputsAddress , outputCount => _outputsCount);
                IF _inputsCount <> UINT#20 OR _outputsCount <> UINT#0 THEN
                    Messenger.Activate(UINT#1116,eAxoMessageCategory#Error);
                    Status.Error.Id := UINT#1116;
                    RETURN;
                END_IF;
                //******************Slot 42*****************//
                _geoAddr.Slot   :=  UINT#42;
                _geoAddr.HardwareType := UINT#4; // (4-Module)
                _retval := ReadHardwareIDFromSlot(geoAddr := _geoAddr, hardwareID => Config.HWIDs.HwID_ToolResult_36);
                IF Config.HWIDs.HwID_ToolResult_36 = UINT#0 THEN
                    Messenger.Activate(UINT#1120,eAxoMessageCategory#Error);
                    Status.Error.Id := UINT#1120;
                    RETURN;
                END_IF;
                IF _retval = WORD#8091 THEN
                    Messenger.Activate(UINT#1121,eAxoMessageCategory#Error);
                    Status.Error.Id := UINT#1121;
                    RETURN;
                END_IF;
                IF _retval = WORD#8094 THEN
                    Messenger.Activate(UINT#1122,eAxoMessageCategory#Error);
                    Status.Error.Id := UINT#1122;
                    RETURN;
                END_IF;
                IF _retval = WORD#8095 THEN
                    Messenger.Activate(UINT#1123,eAxoMessageCategory#Error);
                    Status.Error.Id := UINT#1123;
                    RETURN;
                END_IF;
                IF _retval = WORD#8096 THEN
                    Messenger.Activate(UINT#1124,eAxoMessageCategory#Error);
                    Status.Error.Id := UINT#1124;
                    RETURN;
                END_IF;
                IF _retval = WORD#8097 THEN
                    Messenger.Activate(UINT#1125,eAxoMessageCategory#Error);
                    Status.Error.Id := UINT#1125;
                    RETURN;
                END_IF;
                ReadHardwareIOAddress(hardwareID := (Config.HWIDs.HwID_ToolResult_36) , inputStartAddress => _inputsAddress , inputCount => _inputsCount , outputStartAddress => _outputsAddress , outputCount => _outputsCount);
                IF _inputsCount <> UINT#20 OR _outputsCount <> UINT#0 THEN
                    Messenger.Activate(UINT#1126,eAxoMessageCategory#Error);
                    Status.Error.Id := UINT#1126;
                    RETURN;
                END_IF;
                //******************Slot 43*****************//
                _geoAddr.Slot   :=  UINT#43;
                _geoAddr.HardwareType := UINT#4; // (4-Module)
                _retval := ReadHardwareIDFromSlot(geoAddr := _geoAddr, hardwareID => Config.HWIDs.HwID_ToolResult_37);
                IF Config.HWIDs.HwID_ToolResult_37 = UINT#0 THEN
                    Messenger.Activate(UINT#1130,eAxoMessageCategory#Error);
                    Status.Error.Id := UINT#1130;
                    RETURN;
                END_IF;
                IF _retval = WORD#8091 THEN
                    Messenger.Activate(UINT#1131,eAxoMessageCategory#Error);
                    Status.Error.Id := UINT#1131;
                    RETURN;
                END_IF;
                IF _retval = WORD#8094 THEN
                    Messenger.Activate(UINT#1132,eAxoMessageCategory#Error);
                    Status.Error.Id := UINT#1132;
                    RETURN;
                END_IF;
                IF _retval = WORD#8095 THEN
                    Messenger.Activate(UINT#1133,eAxoMessageCategory#Error);
                    Status.Error.Id := UINT#1133;
                    RETURN;
                END_IF;
                IF _retval = WORD#8096 THEN
                    Messenger.Activate(UINT#1134,eAxoMessageCategory#Error);
                    Status.Error.Id := UINT#1134;
                    RETURN;
                END_IF;
                IF _retval = WORD#8097 THEN
                    Messenger.Activate(UINT#1135,eAxoMessageCategory#Error);
                    Status.Error.Id := UINT#1135;
                    RETURN;
                END_IF;
                ReadHardwareIOAddress(hardwareID := (Config.HWIDs.HwID_ToolResult_37) , inputStartAddress => _inputsAddress , inputCount => _inputsCount , outputStartAddress => _outputsAddress , outputCount => _outputsCount);
                IF _inputsCount <> UINT#20 OR _outputsCount <> UINT#0 THEN
                    Messenger.Activate(UINT#1136,eAxoMessageCategory#Error);
                    Status.Error.Id := UINT#1136;
                    RETURN;
                END_IF;
                //******************Slot 44*****************//
                _geoAddr.Slot   :=  UINT#44;
                _geoAddr.HardwareType := UINT#4; // (4-Module)
                _retval := ReadHardwareIDFromSlot(geoAddr := _geoAddr, hardwareID => Config.HWIDs.HwID_ToolResult_38);
                IF Config.HWIDs.HwID_ToolResult_38 = UINT#0 THEN
                    Messenger.Activate(UINT#1140,eAxoMessageCategory#Error);
                    Status.Error.Id := UINT#1140;
                    RETURN;
                END_IF;
                IF _retval = WORD#8091 THEN
                    Messenger.Activate(UINT#1141,eAxoMessageCategory#Error);
                    Status.Error.Id := UINT#1141;
                    RETURN;
                END_IF;
                IF _retval = WORD#8094 THEN
                    Messenger.Activate(UINT#1142,eAxoMessageCategory#Error);
                    Status.Error.Id := UINT#1142;
                    RETURN;
                END_IF;
                IF _retval = WORD#8095 THEN
                    Messenger.Activate(UINT#1143,eAxoMessageCategory#Error);
                    Status.Error.Id := UINT#1143;
                    RETURN;
                END_IF;
                IF _retval = WORD#8096 THEN
                    Messenger.Activate(UINT#1144,eAxoMessageCategory#Error);
                    Status.Error.Id := UINT#1144;
                    RETURN;
                END_IF;
                IF _retval = WORD#8097 THEN
                    Messenger.Activate(UINT#1145,eAxoMessageCategory#Error);
                    Status.Error.Id := UINT#1145;
                    RETURN;
                END_IF;
                ReadHardwareIOAddress(hardwareID := (Config.HWIDs.HwID_ToolResult_38) , inputStartAddress => _inputsAddress , inputCount => _inputsCount , outputStartAddress => _outputsAddress , outputCount => _outputsCount);
                IF _inputsCount <> UINT#20 OR _outputsCount <> UINT#0 THEN
                    Messenger.Activate(UINT#1146,eAxoMessageCategory#Error);
                    Status.Error.Id := UINT#1146;
                    RETURN;
                END_IF;
                //******************Slot 45*****************//
                _geoAddr.Slot   :=  UINT#45;
                _geoAddr.HardwareType := UINT#4; // (4-Module)
                _retval := ReadHardwareIDFromSlot(geoAddr := _geoAddr, hardwareID => Config.HWIDs.HwID_ToolResult_39);
                IF Config.HWIDs.HwID_ToolResult_39 = UINT#0 THEN
                    Messenger.Activate(UINT#1150,eAxoMessageCategory#Error);
                    Status.Error.Id := UINT#1150;
                    RETURN;
                END_IF;
                IF _retval = WORD#8091 THEN
                    Messenger.Activate(UINT#1151,eAxoMessageCategory#Error);
                    Status.Error.Id := UINT#1151;
                    RETURN;
                END_IF;
                IF _retval = WORD#8094 THEN
                    Messenger.Activate(UINT#1152,eAxoMessageCategory#Error);
                    Status.Error.Id := UINT#1152;
                    RETURN;
                END_IF;
                IF _retval = WORD#8095 THEN
                    Messenger.Activate(UINT#1153,eAxoMessageCategory#Error);
                    Status.Error.Id := UINT#1153;
                    RETURN;
                END_IF;
                IF _retval = WORD#8096 THEN
                    Messenger.Activate(UINT#1154,eAxoMessageCategory#Error);
                    Status.Error.Id := UINT#1154;
                    RETURN;
                END_IF;
                IF _retval = WORD#8097 THEN
                    Messenger.Activate(UINT#1155,eAxoMessageCategory#Error);
                    Status.Error.Id := UINT#1155;
                    RETURN;
                END_IF;
                ReadHardwareIOAddress(hardwareID := (Config.HWIDs.HwID_ToolResult_39) , inputStartAddress => _inputsAddress , inputCount => _inputsCount , outputStartAddress => _outputsAddress , outputCount => _outputsCount);
                IF _inputsCount <> UINT#20 OR _outputsCount <> UINT#0 THEN
                    Messenger.Activate(UINT#1156,eAxoMessageCategory#Error);
                    Status.Error.Id := UINT#1156;
                    RETURN;
                END_IF;
                //******************Slot 46*****************//
                _geoAddr.Slot   :=  UINT#46;
                _geoAddr.HardwareType := UINT#4; // (4-Module)
                _retval := ReadHardwareIDFromSlot(geoAddr := _geoAddr, hardwareID => Config.HWIDs.HwID_ToolResult_40);
                IF Config.HWIDs.HwID_ToolResult_40 = UINT#0 THEN
                    Messenger.Activate(UINT#1160,eAxoMessageCategory#Error);
                    Status.Error.Id := UINT#1160;
                    RETURN;
                END_IF;
                IF _retval = WORD#8091 THEN
                    Messenger.Activate(UINT#1161,eAxoMessageCategory#Error);
                    Status.Error.Id := UINT#1161;
                    RETURN;
                END_IF;
                IF _retval = WORD#8094 THEN
                    Messenger.Activate(UINT#1162,eAxoMessageCategory#Error);
                    Status.Error.Id := UINT#1162;
                    RETURN;
                END_IF;
                IF _retval = WORD#8095 THEN
                    Messenger.Activate(UINT#1163,eAxoMessageCategory#Error);
                    Status.Error.Id := UINT#1163;
                    RETURN;
                END_IF;
                IF _retval = WORD#8096 THEN
                    Messenger.Activate(UINT#1164,eAxoMessageCategory#Error);
                    Status.Error.Id := UINT#1164;
                    RETURN;
                END_IF;
                IF _retval = WORD#8097 THEN
                    Messenger.Activate(UINT#1165,eAxoMessageCategory#Error);
                    Status.Error.Id := UINT#1165;
                    RETURN;
                END_IF;
                ReadHardwareIOAddress(hardwareID := (Config.HWIDs.HwID_ToolResult_40) , inputStartAddress => _inputsAddress , inputCount => _inputsCount , outputStartAddress => _outputsAddress , outputCount => _outputsCount);
                IF _inputsCount <> UINT#20 OR _outputsCount <> UINT#0 THEN
                    Messenger.Activate(UINT#1166,eAxoMessageCategory#Error);
                    Status.Error.Id := UINT#1166;
                    RETURN;
                END_IF;
                //******************Slot 47*****************//
                _geoAddr.Slot   :=  UINT#47;
                _geoAddr.HardwareType := UINT#4; // (4-Module)
                _retval := ReadHardwareIDFromSlot(geoAddr := _geoAddr, hardwareID => Config.HWIDs.HwID_ToolResult_41);
                IF Config.HWIDs.HwID_ToolResult_41 = UINT#0 THEN
                    Messenger.Activate(UINT#1170,eAxoMessageCategory#Error);
                    Status.Error.Id := UINT#1170;
                    RETURN;
                END_IF;
                IF _retval = WORD#8091 THEN
                    Messenger.Activate(UINT#1171,eAxoMessageCategory#Error);
                    Status.Error.Id := UINT#1171;
                    RETURN;
                END_IF;
                IF _retval = WORD#8094 THEN
                    Messenger.Activate(UINT#1172,eAxoMessageCategory#Error);
                    Status.Error.Id := UINT#1172;
                    RETURN;
                END_IF;
                IF _retval = WORD#8095 THEN
                    Messenger.Activate(UINT#1173,eAxoMessageCategory#Error);
                    Status.Error.Id := UINT#1173;
                    RETURN;
                END_IF;
                IF _retval = WORD#8096 THEN
                    Messenger.Activate(UINT#1174,eAxoMessageCategory#Error);
                    Status.Error.Id := UINT#1174;
                    RETURN;
                END_IF;
                IF _retval = WORD#8097 THEN
                    Messenger.Activate(UINT#1175,eAxoMessageCategory#Error);
                    Status.Error.Id := UINT#1175;
                    RETURN;
                END_IF;
                ReadHardwareIOAddress(hardwareID := (Config.HWIDs.HwID_ToolResult_41) , inputStartAddress => _inputsAddress , inputCount => _inputsCount , outputStartAddress => _outputsAddress , outputCount => _outputsCount);
                IF _inputsCount <> UINT#20 OR _outputsCount <> UINT#0 THEN
                    Messenger.Activate(UINT#1176,eAxoMessageCategory#Error);
                    Status.Error.Id := UINT#1176;
                    RETURN;
                END_IF;
                //******************Slot 48*****************//
                _geoAddr.Slot   :=  UINT#48;
                _geoAddr.HardwareType := UINT#4; // (4-Module)
                _retval := ReadHardwareIDFromSlot(geoAddr := _geoAddr, hardwareID => Config.HWIDs.HwID_ToolResult_42);
                IF Config.HWIDs.HwID_ToolResult_42 = UINT#0 THEN
                    Messenger.Activate(UINT#1180,eAxoMessageCategory#Error);
                    Status.Error.Id := UINT#1180;
                    RETURN;
                END_IF;
                IF _retval = WORD#8091 THEN
                    Messenger.Activate(UINT#1181,eAxoMessageCategory#Error);
                    Status.Error.Id := UINT#1181;
                    RETURN;
                END_IF;
                IF _retval = WORD#8094 THEN
                    Messenger.Activate(UINT#1182,eAxoMessageCategory#Error);
                    Status.Error.Id := UINT#1182;
                    RETURN;
                END_IF;
                IF _retval = WORD#8095 THEN
                    Messenger.Activate(UINT#1183,eAxoMessageCategory#Error);
                    Status.Error.Id := UINT#1183;
                    RETURN;
                END_IF;
                IF _retval = WORD#8096 THEN
                    Messenger.Activate(UINT#1184,eAxoMessageCategory#Error);
                    Status.Error.Id := UINT#1184;
                    RETURN;
                END_IF;
                IF _retval = WORD#8097 THEN
                    Messenger.Activate(UINT#1185,eAxoMessageCategory#Error);
                    Status.Error.Id := UINT#1185;
                    RETURN;
                END_IF;
                ReadHardwareIOAddress(hardwareID := (Config.HWIDs.HwID_ToolResult_42) , inputStartAddress => _inputsAddress , inputCount => _inputsCount , outputStartAddress => _outputsAddress , outputCount => _outputsCount);
                IF _inputsCount <> UINT#20 OR _outputsCount <> UINT#0 THEN
                    Messenger.Activate(UINT#1186,eAxoMessageCategory#Error);
                    Status.Error.Id := UINT#1186;
                    RETURN;
                END_IF;
                //******************Slot 49*****************//
                _geoAddr.Slot   :=  UINT#49;
                _geoAddr.HardwareType := UINT#4; // (4-Module)
                _retval := ReadHardwareIDFromSlot(geoAddr := _geoAddr, hardwareID => Config.HWIDs.HwID_ToolResult_43);
                IF Config.HWIDs.HwID_ToolResult_43 = UINT#0 THEN
                    Messenger.Activate(UINT#1190,eAxoMessageCategory#Error);
                    Status.Error.Id := UINT#1190;
                    RETURN;
                END_IF;
                IF _retval = WORD#8091 THEN
                    Messenger.Activate(UINT#1191,eAxoMessageCategory#Error);
                    Status.Error.Id := UINT#1191;
                    RETURN;
                END_IF;
                IF _retval = WORD#8094 THEN
                    Messenger.Activate(UINT#1192,eAxoMessageCategory#Error);
                    Status.Error.Id := UINT#1192;
                    RETURN;
                END_IF;
                IF _retval = WORD#8095 THEN
                    Messenger.Activate(UINT#1193,eAxoMessageCategory#Error);
                    Status.Error.Id := UINT#1193;
                    RETURN;
                END_IF;
                IF _retval = WORD#8096 THEN
                    Messenger.Activate(UINT#1194,eAxoMessageCategory#Error);
                    Status.Error.Id := UINT#1194;
                    RETURN;
                END_IF;
                IF _retval = WORD#8097 THEN
                    Messenger.Activate(UINT#1195,eAxoMessageCategory#Error);
                    Status.Error.Id := UINT#1195;
                    RETURN;
                END_IF;
                ReadHardwareIOAddress(hardwareID := (Config.HWIDs.HwID_ToolResult_43) , inputStartAddress => _inputsAddress , inputCount => _inputsCount , outputStartAddress => _outputsAddress , outputCount => _outputsCount);
                IF _inputsCount <> UINT#20 OR _outputsCount <> UINT#0 THEN
                    Messenger.Activate(UINT#1196,eAxoMessageCategory#Error);
                    Status.Error.Id := UINT#1196;
                    RETURN;
                END_IF;
                //******************Slot 50*****************//
                _geoAddr.Slot   :=  UINT#50;
                _geoAddr.HardwareType := UINT#4; // (4-Module)
                _retval := ReadHardwareIDFromSlot(geoAddr := _geoAddr, hardwareID => Config.HWIDs.HwID_ToolResult_44);
                IF Config.HWIDs.HwID_ToolResult_44 = UINT#0 THEN
                    Messenger.Activate(UINT#1200,eAxoMessageCategory#Error);
                    Status.Error.Id := UINT#1200;
                    RETURN;
                END_IF;
                IF _retval = WORD#8091 THEN
                    Messenger.Activate(UINT#1201,eAxoMessageCategory#Error);
                    Status.Error.Id := UINT#1201;
                    RETURN;
                END_IF;
                IF _retval = WORD#8094 THEN
                    Messenger.Activate(UINT#1202,eAxoMessageCategory#Error);
                    Status.Error.Id := UINT#1202;
                    RETURN;
                END_IF;
                IF _retval = WORD#8095 THEN
                    Messenger.Activate(UINT#1203,eAxoMessageCategory#Error);
                    Status.Error.Id := UINT#1203;
                    RETURN;
                END_IF;
                IF _retval = WORD#8096 THEN
                    Messenger.Activate(UINT#1204,eAxoMessageCategory#Error);
                    Status.Error.Id := UINT#1204;
                    RETURN;
                END_IF;
                IF _retval = WORD#8097 THEN
                    Messenger.Activate(UINT#1205,eAxoMessageCategory#Error);
                    Status.Error.Id := UINT#1205;
                    RETURN;
                END_IF;
                ReadHardwareIOAddress(hardwareID := (Config.HWIDs.HwID_ToolResult_44) , inputStartAddress => _inputsAddress , inputCount => _inputsCount , outputStartAddress => _outputsAddress , outputCount => _outputsCount);
                IF _inputsCount <> UINT#20 OR _outputsCount <> UINT#0 THEN
                    Messenger.Activate(UINT#1206,eAxoMessageCategory#Error);
                    Status.Error.Id := UINT#1206;
                    RETURN;
                END_IF;
                //******************Slot 51*****************//
                _geoAddr.Slot   :=  UINT#51;
                _geoAddr.HardwareType := UINT#4; // (4-Module)
                _retval := ReadHardwareIDFromSlot(geoAddr := _geoAddr, hardwareID => Config.HWIDs.HwID_ToolResult_45);
                IF Config.HWIDs.HwID_ToolResult_45 = UINT#0 THEN
                    Messenger.Activate(UINT#1210,eAxoMessageCategory#Error);
                    Status.Error.Id := UINT#1210;
                    RETURN;
                END_IF;
                IF _retval = WORD#8091 THEN
                    Messenger.Activate(UINT#1211,eAxoMessageCategory#Error);
                    Status.Error.Id := UINT#1211;
                    RETURN;
                END_IF;
                IF _retval = WORD#8094 THEN
                    Messenger.Activate(UINT#1212,eAxoMessageCategory#Error);
                    Status.Error.Id := UINT#1212;
                    RETURN;
                END_IF;
                IF _retval = WORD#8095 THEN
                    Messenger.Activate(UINT#1213,eAxoMessageCategory#Error);
                    Status.Error.Id := UINT#1213;
                    RETURN;
                END_IF;
                IF _retval = WORD#8096 THEN
                    Messenger.Activate(UINT#1214,eAxoMessageCategory#Error);
                    Status.Error.Id := UINT#1214;
                    RETURN;
                END_IF;
                IF _retval = WORD#8097 THEN
                    Messenger.Activate(UINT#1215,eAxoMessageCategory#Error);
                    Status.Error.Id := UINT#1215;
                    RETURN;
                END_IF;
                ReadHardwareIOAddress(hardwareID := (Config.HWIDs.HwID_ToolResult_45) , inputStartAddress => _inputsAddress , inputCount => _inputsCount , outputStartAddress => _outputsAddress , outputCount => _outputsCount);
                IF _inputsCount <> UINT#20 OR _outputsCount <> UINT#0 THEN
                    Messenger.Activate(UINT#1216,eAxoMessageCategory#Error);
                    Status.Error.Id := UINT#1216;
                    RETURN;
                END_IF;
                //******************Slot 52*****************//
                _geoAddr.Slot   :=  UINT#52;
                _geoAddr.HardwareType := UINT#4; // (4-Module)
                _retval := ReadHardwareIDFromSlot(geoAddr := _geoAddr, hardwareID => Config.HWIDs.HwID_ToolResult_46);
                IF Config.HWIDs.HwID_ToolResult_46 = UINT#0 THEN
                    Messenger.Activate(UINT#1220,eAxoMessageCategory#Error);
                    Status.Error.Id := UINT#1220;
                    RETURN;
                END_IF;
                IF _retval = WORD#8091 THEN
                    Messenger.Activate(UINT#1221,eAxoMessageCategory#Error);
                    Status.Error.Id := UINT#1221;
                    RETURN;
                END_IF;
                IF _retval = WORD#8094 THEN
                    Messenger.Activate(UINT#1222,eAxoMessageCategory#Error);
                    Status.Error.Id := UINT#1222;
                    RETURN;
                END_IF;
                IF _retval = WORD#8095 THEN
                    Messenger.Activate(UINT#1223,eAxoMessageCategory#Error);
                    Status.Error.Id := UINT#1223;
                    RETURN;
                END_IF;
                IF _retval = WORD#8096 THEN
                    Messenger.Activate(UINT#1224,eAxoMessageCategory#Error);
                    Status.Error.Id := UINT#1224;
                    RETURN;
                END_IF;
                IF _retval = WORD#8097 THEN
                    Messenger.Activate(UINT#1225,eAxoMessageCategory#Error);
                    Status.Error.Id := UINT#1225;
                    RETURN;
                END_IF;
                ReadHardwareIOAddress(hardwareID := (Config.HWIDs.HwID_ToolResult_46) , inputStartAddress => _inputsAddress , inputCount => _inputsCount , outputStartAddress => _outputsAddress , outputCount => _outputsCount);
                IF _inputsCount <> UINT#20 OR _outputsCount <> UINT#0 THEN
                    Messenger.Activate(UINT#1226,eAxoMessageCategory#Error);
                    Status.Error.Id := UINT#1226;
                    RETURN;
                END_IF;
                //******************Slot 53*****************//
                _geoAddr.Slot   :=  UINT#53;
                _geoAddr.HardwareType := UINT#4; // (4-Module)
                _retval := ReadHardwareIDFromSlot(geoAddr := _geoAddr, hardwareID => Config.HWIDs.HwID_ToolResult_47);
                IF Config.HWIDs.HwID_ToolResult_47 = UINT#0 THEN
                    Messenger.Activate(UINT#1230,eAxoMessageCategory#Error);
                    Status.Error.Id := UINT#1230;
                    RETURN;
                END_IF;
                IF _retval = WORD#8091 THEN
                    Messenger.Activate(UINT#1231,eAxoMessageCategory#Error);
                    Status.Error.Id := UINT#1231;
                    RETURN;
                END_IF;
                IF _retval = WORD#8094 THEN
                    Messenger.Activate(UINT#1232,eAxoMessageCategory#Error);
                    Status.Error.Id := UINT#1232;
                    RETURN;
                END_IF;
                IF _retval = WORD#8095 THEN
                    Messenger.Activate(UINT#1233,eAxoMessageCategory#Error);
                    Status.Error.Id := UINT#1233;
                    RETURN;
                END_IF;
                IF _retval = WORD#8096 THEN
                    Messenger.Activate(UINT#1234,eAxoMessageCategory#Error);
                    Status.Error.Id := UINT#1234;
                    RETURN;
                END_IF;
                IF _retval = WORD#8097 THEN
                    Messenger.Activate(UINT#1235,eAxoMessageCategory#Error);
                    Status.Error.Id := UINT#1235;
                    RETURN;
                END_IF;
                ReadHardwareIOAddress(hardwareID := (Config.HWIDs.HwID_ToolResult_47) , inputStartAddress => _inputsAddress , inputCount => _inputsCount , outputStartAddress => _outputsAddress , outputCount => _outputsCount);
                IF _inputsCount <> UINT#20 OR _outputsCount <> UINT#0 THEN
                    Messenger.Activate(UINT#1236,eAxoMessageCategory#Error);
                    Status.Error.Id := UINT#1236;
                    RETURN;
                END_IF;
                //******************Slot 54*****************//
                _geoAddr.Slot   :=  UINT#54;
                _geoAddr.HardwareType := UINT#4; // (4-Module)
                _retval := ReadHardwareIDFromSlot(geoAddr := _geoAddr, hardwareID => Config.HWIDs.HwID_ToolResult_48);
                IF Config.HWIDs.HwID_ToolResult_48 = UINT#0 THEN
                    Messenger.Activate(UINT#1240,eAxoMessageCategory#Error);
                    Status.Error.Id := UINT#1240;
                    RETURN;
                END_IF;
                IF _retval = WORD#8091 THEN
                    Messenger.Activate(UINT#1241,eAxoMessageCategory#Error);
                    Status.Error.Id := UINT#1241;
                    RETURN;
                END_IF;
                IF _retval = WORD#8094 THEN
                    Messenger.Activate(UINT#1242,eAxoMessageCategory#Error);
                    Status.Error.Id := UINT#1242;
                    RETURN;
                END_IF;
                IF _retval = WORD#8095 THEN
                    Messenger.Activate(UINT#1243,eAxoMessageCategory#Error);
                    Status.Error.Id := UINT#1243;
                    RETURN;
                END_IF;
                IF _retval = WORD#8096 THEN
                    Messenger.Activate(UINT#1244,eAxoMessageCategory#Error);
                    Status.Error.Id := UINT#1244;
                    RETURN;
                END_IF;
                IF _retval = WORD#8097 THEN
                    Messenger.Activate(UINT#1245,eAxoMessageCategory#Error);
                    Status.Error.Id := UINT#1245;
                    RETURN;
                END_IF;
                ReadHardwareIOAddress(hardwareID := (Config.HWIDs.HwID_ToolResult_48) , inputStartAddress => _inputsAddress , inputCount => _inputsCount , outputStartAddress => _outputsAddress , outputCount => _outputsCount);
                IF _inputsCount <> UINT#20 OR _outputsCount <> UINT#0 THEN
                    Messenger.Activate(UINT#1246,eAxoMessageCategory#Error);
                    Status.Error.Id := UINT#1246;
                    RETURN;
                END_IF;
                //******************Slot 55*****************//
                _geoAddr.Slot   :=  UINT#55;
                _geoAddr.HardwareType := UINT#4; // (4-Module)
                _retval := ReadHardwareIDFromSlot(geoAddr := _geoAddr, hardwareID => Config.HWIDs.HwID_ToolResult_49);
                IF Config.HWIDs.HwID_ToolResult_49 = UINT#0 THEN
                    Messenger.Activate(UINT#1250,eAxoMessageCategory#Error);
                    Status.Error.Id := UINT#1250;
                    RETURN;
                END_IF;
                IF _retval = WORD#8091 THEN
                    Messenger.Activate(UINT#1251,eAxoMessageCategory#Error);
                    Status.Error.Id := UINT#1251;
                    RETURN;
                END_IF;
                IF _retval = WORD#8094 THEN
                    Messenger.Activate(UINT#1252,eAxoMessageCategory#Error);
                    Status.Error.Id := UINT#1252;
                    RETURN;
                END_IF;
                IF _retval = WORD#8095 THEN
                    Messenger.Activate(UINT#1253,eAxoMessageCategory#Error);
                    Status.Error.Id := UINT#1253;
                    RETURN;
                END_IF;
                IF _retval = WORD#8096 THEN
                    Messenger.Activate(UINT#1254,eAxoMessageCategory#Error);
                    Status.Error.Id := UINT#1254;
                    RETURN;
                END_IF;
                IF _retval = WORD#8097 THEN
                    Messenger.Activate(UINT#1255,eAxoMessageCategory#Error);
                    Status.Error.Id := UINT#1255;
                    RETURN;
                END_IF;
                ReadHardwareIOAddress(hardwareID := (Config.HWIDs.HwID_ToolResult_49) , inputStartAddress => _inputsAddress , inputCount => _inputsCount , outputStartAddress => _outputsAddress , outputCount => _outputsCount);
                IF _inputsCount <> UINT#20 OR _outputsCount <> UINT#0 THEN
                    Messenger.Activate(UINT#1256,eAxoMessageCategory#Error);
                    Status.Error.Id := UINT#1256;
                    RETURN;
                END_IF;
                //******************Slot 56*****************//
                _geoAddr.Slot   :=  UINT#56;
                _geoAddr.HardwareType := UINT#4; // (4-Module)
                _retval := ReadHardwareIDFromSlot(geoAddr := _geoAddr, hardwareID => Config.HWIDs.HwID_ToolResult_50);
                IF Config.HWIDs.HwID_ToolResult_50 = UINT#0 THEN
                    Messenger.Activate(UINT#1260,eAxoMessageCategory#Error);
                    Status.Error.Id := UINT#1260;
                    RETURN;
                END_IF;
                IF _retval = WORD#8091 THEN
                    Messenger.Activate(UINT#1261,eAxoMessageCategory#Error);
                    Status.Error.Id := UINT#1261;
                    RETURN;
                END_IF;
                IF _retval = WORD#8094 THEN
                    Messenger.Activate(UINT#1262,eAxoMessageCategory#Error);
                    Status.Error.Id := UINT#1262;
                    RETURN;
                END_IF;
                IF _retval = WORD#8095 THEN
                    Messenger.Activate(UINT#1263,eAxoMessageCategory#Error);
                    Status.Error.Id := UINT#1263;
                    RETURN;
                END_IF;
                IF _retval = WORD#8096 THEN
                    Messenger.Activate(UINT#1264,eAxoMessageCategory#Error);
                    Status.Error.Id := UINT#1264;
                    RETURN;
                END_IF;
                IF _retval = WORD#8097 THEN
                    Messenger.Activate(UINT#1265,eAxoMessageCategory#Error);
                    Status.Error.Id := UINT#1265;
                    RETURN;
                END_IF;
                ReadHardwareIOAddress(hardwareID := (Config.HWIDs.HwID_ToolResult_50) , inputStartAddress => _inputsAddress , inputCount => _inputsCount , outputStartAddress => _outputsAddress , outputCount => _outputsCount);
                IF _inputsCount <> UINT#20 OR _outputsCount <> UINT#0 THEN
                    Messenger.Activate(UINT#1266,eAxoMessageCategory#Error);
                    Status.Error.Id := UINT#1266;
                    RETURN;
                END_IF;
                //******************Slot 57*****************//
                _geoAddr.Slot   :=  UINT#57;
                _geoAddr.HardwareType := UINT#4; // (4-Module)
                _retval := ReadHardwareIDFromSlot(geoAddr := _geoAddr, hardwareID => Config.HWIDs.HwID_ToolResult_51);
                IF Config.HWIDs.HwID_ToolResult_51 = UINT#0 THEN
                    Messenger.Activate(UINT#1270,eAxoMessageCategory#Error);
                    Status.Error.Id := UINT#1270;
                    RETURN;
                END_IF;
                IF _retval = WORD#8091 THEN
                    Messenger.Activate(UINT#1271,eAxoMessageCategory#Error);
                    Status.Error.Id := UINT#1271;
                    RETURN;
                END_IF;
                IF _retval = WORD#8094 THEN
                    Messenger.Activate(UINT#1272,eAxoMessageCategory#Error);
                    Status.Error.Id := UINT#1272;
                    RETURN;
                END_IF;
                IF _retval = WORD#8095 THEN
                    Messenger.Activate(UINT#1273,eAxoMessageCategory#Error);
                    Status.Error.Id := UINT#1273;
                    RETURN;
                END_IF;
                IF _retval = WORD#8096 THEN
                    Messenger.Activate(UINT#1274,eAxoMessageCategory#Error);
                    Status.Error.Id := UINT#1274;
                    RETURN;
                END_IF;
                IF _retval = WORD#8097 THEN
                    Messenger.Activate(UINT#1275,eAxoMessageCategory#Error);
                    Status.Error.Id := UINT#1275;
                    RETURN;
                END_IF;
                ReadHardwareIOAddress(hardwareID := (Config.HWIDs.HwID_ToolResult_51) , inputStartAddress => _inputsAddress , inputCount => _inputsCount , outputStartAddress => _outputsAddress , outputCount => _outputsCount);
                IF _inputsCount <> UINT#20 OR _outputsCount <> UINT#0 THEN
                    Messenger.Activate(UINT#1276,eAxoMessageCategory#Error);
                    Status.Error.Id := UINT#1276;
                    RETURN;
                END_IF;
                //******************Slot 58*****************//
                _geoAddr.Slot   :=  UINT#58;
                _geoAddr.HardwareType := UINT#4; // (4-Module)
                _retval := ReadHardwareIDFromSlot(geoAddr := _geoAddr, hardwareID => Config.HWIDs.HwID_ToolResult_52);
                IF Config.HWIDs.HwID_ToolResult_52 = UINT#0 THEN
                    Messenger.Activate(UINT#1280,eAxoMessageCategory#Error);
                    Status.Error.Id := UINT#1280;
                    RETURN;
                END_IF;
                IF _retval = WORD#8091 THEN
                    Messenger.Activate(UINT#1281,eAxoMessageCategory#Error);
                    Status.Error.Id := UINT#1281;
                    RETURN;
                END_IF;
                IF _retval = WORD#8094 THEN
                    Messenger.Activate(UINT#1282,eAxoMessageCategory#Error);
                    Status.Error.Id := UINT#1282;
                    RETURN;
                END_IF;
                IF _retval = WORD#8095 THEN
                    Messenger.Activate(UINT#1283,eAxoMessageCategory#Error);
                    Status.Error.Id := UINT#1283;
                    RETURN;
                END_IF;
                IF _retval = WORD#8096 THEN
                    Messenger.Activate(UINT#1284,eAxoMessageCategory#Error);
                    Status.Error.Id := UINT#1284;
                    RETURN;
                END_IF;
                IF _retval = WORD#8097 THEN
                    Messenger.Activate(UINT#1285,eAxoMessageCategory#Error);
                    Status.Error.Id := UINT#1285;
                    RETURN;
                END_IF;
                ReadHardwareIOAddress(hardwareID := (Config.HWIDs.HwID_ToolResult_52) , inputStartAddress => _inputsAddress , inputCount => _inputsCount , outputStartAddress => _outputsAddress , outputCount => _outputsCount);
                IF _inputsCount <> UINT#20 OR _outputsCount <> UINT#0 THEN
                    Messenger.Activate(UINT#1286,eAxoMessageCategory#Error);
                    Status.Error.Id := UINT#1286;
                    RETURN;
                END_IF;
                //******************Slot 59*****************//
                _geoAddr.Slot   :=  UINT#59;
                _geoAddr.HardwareType := UINT#4; // (4-Module)
                _retval := ReadHardwareIDFromSlot(geoAddr := _geoAddr, hardwareID => Config.HWIDs.HwID_ToolResult_53);
                IF Config.HWIDs.HwID_ToolResult_53 = UINT#0 THEN
                    Messenger.Activate(UINT#1290,eAxoMessageCategory#Error);
                    Status.Error.Id := UINT#1290;
                    RETURN;
                END_IF;
                IF _retval = WORD#8091 THEN
                    Messenger.Activate(UINT#1291,eAxoMessageCategory#Error);
                    Status.Error.Id := UINT#1291;
                    RETURN;
                END_IF;
                IF _retval = WORD#8094 THEN
                    Messenger.Activate(UINT#1292,eAxoMessageCategory#Error);
                    Status.Error.Id := UINT#1292;
                    RETURN;
                END_IF;
                IF _retval = WORD#8095 THEN
                    Messenger.Activate(UINT#1293,eAxoMessageCategory#Error);
                    Status.Error.Id := UINT#1293;
                    RETURN;
                END_IF;
                IF _retval = WORD#8096 THEN
                    Messenger.Activate(UINT#1294,eAxoMessageCategory#Error);
                    Status.Error.Id := UINT#1294;
                    RETURN;
                END_IF;
                IF _retval = WORD#8097 THEN
                    Messenger.Activate(UINT#1295,eAxoMessageCategory#Error);
                    Status.Error.Id := UINT#1295;
                    RETURN;
                END_IF;
                ReadHardwareIOAddress(hardwareID := (Config.HWIDs.HwID_ToolResult_53) , inputStartAddress => _inputsAddress , inputCount => _inputsCount , outputStartAddress => _outputsAddress , outputCount => _outputsCount);
                IF _inputsCount <> UINT#20 OR _outputsCount <> UINT#0 THEN
                    Messenger.Activate(UINT#1296,eAxoMessageCategory#Error);
                    Status.Error.Id := UINT#1296;
                    RETURN;
                END_IF;
                //******************Slot 60*****************//
                _geoAddr.Slot   :=  UINT#60;
                _geoAddr.HardwareType := UINT#4; // (4-Module)
                _retval := ReadHardwareIDFromSlot(geoAddr := _geoAddr, hardwareID => Config.HWIDs.HwID_ToolResult_54);
                IF Config.HWIDs.HwID_ToolResult_54 = UINT#0 THEN
                    Messenger.Activate(UINT#1300,eAxoMessageCategory#Error);
                    Status.Error.Id := UINT#1300;
                    RETURN;
                END_IF;
                IF _retval = WORD#8091 THEN
                    Messenger.Activate(UINT#1301,eAxoMessageCategory#Error);
                    Status.Error.Id := UINT#1301;
                    RETURN;
                END_IF;
                IF _retval = WORD#8094 THEN
                    Messenger.Activate(UINT#1302,eAxoMessageCategory#Error);
                    Status.Error.Id := UINT#1302;
                    RETURN;
                END_IF;
                IF _retval = WORD#8095 THEN
                    Messenger.Activate(UINT#1303,eAxoMessageCategory#Error);
                    Status.Error.Id := UINT#1303;
                    RETURN;
                END_IF;
                IF _retval = WORD#8096 THEN
                    Messenger.Activate(UINT#1304,eAxoMessageCategory#Error);
                    Status.Error.Id := UINT#1304;
                    RETURN;
                END_IF;
                IF _retval = WORD#8097 THEN
                    Messenger.Activate(UINT#1305,eAxoMessageCategory#Error);
                    Status.Error.Id := UINT#1305;
                    RETURN;
                END_IF;
                ReadHardwareIOAddress(hardwareID := (Config.HWIDs.HwID_ToolResult_54) , inputStartAddress => _inputsAddress , inputCount => _inputsCount , outputStartAddress => _outputsAddress , outputCount => _outputsCount);
                IF _inputsCount <> UINT#20 OR _outputsCount <> UINT#0 THEN
                    Messenger.Activate(UINT#1306,eAxoMessageCategory#Error);
                    Status.Error.Id := UINT#1306;
                    RETURN;
                END_IF;
                //******************Slot 61*****************//
                _geoAddr.Slot   :=  UINT#61;
                _geoAddr.HardwareType := UINT#4; // (4-Module)
                _retval := ReadHardwareIDFromSlot(geoAddr := _geoAddr, hardwareID => Config.HWIDs.HwID_ToolResult_55);
                IF Config.HWIDs.HwID_ToolResult_55 = UINT#0 THEN
                    Messenger.Activate(UINT#1310,eAxoMessageCategory#Error);
                    Status.Error.Id := UINT#1310;
                    RETURN;
                END_IF;
                IF _retval = WORD#8091 THEN
                    Messenger.Activate(UINT#1311,eAxoMessageCategory#Error);
                    Status.Error.Id := UINT#1311;
                    RETURN;
                END_IF;
                IF _retval = WORD#8094 THEN
                    Messenger.Activate(UINT#1312,eAxoMessageCategory#Error);
                    Status.Error.Id := UINT#1312;
                    RETURN;
                END_IF;
                IF _retval = WORD#8095 THEN
                    Messenger.Activate(UINT#1313,eAxoMessageCategory#Error);
                    Status.Error.Id := UINT#1313;
                    RETURN;
                END_IF;
                IF _retval = WORD#8096 THEN
                    Messenger.Activate(UINT#1314,eAxoMessageCategory#Error);
                    Status.Error.Id := UINT#1314;
                    RETURN;
                END_IF;
                IF _retval = WORD#8097 THEN
                    Messenger.Activate(UINT#1315,eAxoMessageCategory#Error);
                    Status.Error.Id := UINT#1315;
                    RETURN;
                END_IF;
                ReadHardwareIOAddress(hardwareID := (Config.HWIDs.HwID_ToolResult_55) , inputStartAddress => _inputsAddress , inputCount => _inputsCount , outputStartAddress => _outputsAddress , outputCount => _outputsCount);
                IF _inputsCount <> UINT#20 OR _outputsCount <> UINT#0 THEN
                    Messenger.Activate(UINT#1316,eAxoMessageCategory#Error);
                    Status.Error.Id := UINT#1316;
                    RETURN;
                END_IF;
                //******************Slot 62*****************//
                _geoAddr.Slot   :=  UINT#62;
                _geoAddr.HardwareType := UINT#4; // (4-Module)
                _retval := ReadHardwareIDFromSlot(geoAddr := _geoAddr, hardwareID => Config.HWIDs.HwID_ToolResult_56);
                IF Config.HWIDs.HwID_ToolResult_56 = UINT#0 THEN
                    Messenger.Activate(UINT#1320,eAxoMessageCategory#Error);
                    Status.Error.Id := UINT#1320;
                    RETURN;
                END_IF;
                IF _retval = WORD#8091 THEN
                    Messenger.Activate(UINT#1321,eAxoMessageCategory#Error);
                    Status.Error.Id := UINT#1321;
                    RETURN;
                END_IF;
                IF _retval = WORD#8094 THEN
                    Messenger.Activate(UINT#1322,eAxoMessageCategory#Error);
                    Status.Error.Id := UINT#1322;
                    RETURN;
                END_IF;
                IF _retval = WORD#8095 THEN
                    Messenger.Activate(UINT#1323,eAxoMessageCategory#Error);
                    Status.Error.Id := UINT#1323;
                    RETURN;
                END_IF;
                IF _retval = WORD#8096 THEN
                    Messenger.Activate(UINT#1324,eAxoMessageCategory#Error);
                    Status.Error.Id := UINT#1324;
                    RETURN;
                END_IF;
                IF _retval = WORD#8097 THEN
                    Messenger.Activate(UINT#1325,eAxoMessageCategory#Error);
                    Status.Error.Id := UINT#1325;
                    RETURN;
                END_IF;
                ReadHardwareIOAddress(hardwareID := (Config.HWIDs.HwID_ToolResult_56) , inputStartAddress => _inputsAddress , inputCount => _inputsCount , outputStartAddress => _outputsAddress , outputCount => _outputsCount);
                IF _inputsCount <> UINT#20 OR _outputsCount <> UINT#0 THEN
                    Messenger.Activate(UINT#1326,eAxoMessageCategory#Error);
                    Status.Error.Id := UINT#1326;
                    RETURN;
                END_IF;
                //******************Slot 63*****************//
                _geoAddr.Slot   :=  UINT#63;
                _geoAddr.HardwareType := UINT#4; // (4-Module)
                _retval := ReadHardwareIDFromSlot(geoAddr := _geoAddr, hardwareID => Config.HWIDs.HwID_ToolResult_57);
                IF Config.HWIDs.HwID_ToolResult_57 = UINT#0 THEN
                    Messenger.Activate(UINT#1330,eAxoMessageCategory#Error);
                    Status.Error.Id := UINT#1330;
                    RETURN;
                END_IF;
                IF _retval = WORD#8091 THEN
                    Messenger.Activate(UINT#1331,eAxoMessageCategory#Error);
                    Status.Error.Id := UINT#1331;
                    RETURN;
                END_IF;
                IF _retval = WORD#8094 THEN
                    Messenger.Activate(UINT#1332,eAxoMessageCategory#Error);
                    Status.Error.Id := UINT#1332;
                    RETURN;
                END_IF;
                IF _retval = WORD#8095 THEN
                    Messenger.Activate(UINT#1333,eAxoMessageCategory#Error);
                    Status.Error.Id := UINT#1333;
                    RETURN;
                END_IF;
                IF _retval = WORD#8096 THEN
                    Messenger.Activate(UINT#1334,eAxoMessageCategory#Error);
                    Status.Error.Id := UINT#1334;
                    RETURN;
                END_IF;
                IF _retval = WORD#8097 THEN
                    Messenger.Activate(UINT#1335,eAxoMessageCategory#Error);
                    Status.Error.Id := UINT#1335;
                    RETURN;
                END_IF;
                ReadHardwareIOAddress(hardwareID := (Config.HWIDs.HwID_ToolResult_57) , inputStartAddress => _inputsAddress , inputCount => _inputsCount , outputStartAddress => _outputsAddress , outputCount => _outputsCount);
                IF _inputsCount <> UINT#20 OR _outputsCount <> UINT#0 THEN
                    Messenger.Activate(UINT#1336,eAxoMessageCategory#Error);
                    Status.Error.Id := UINT#1336;
                    RETURN;
                END_IF;
                //******************Slot 64*****************//
                _geoAddr.Slot   :=  UINT#64;
                _geoAddr.HardwareType := UINT#4; // (4-Module)
                _retval := ReadHardwareIDFromSlot(geoAddr := _geoAddr, hardwareID => Config.HWIDs.HwID_ToolResult_58);
                IF Config.HWIDs.HwID_ToolResult_58 = UINT#0 THEN
                    Messenger.Activate(UINT#1340,eAxoMessageCategory#Error);
                    Status.Error.Id := UINT#1340;
                    RETURN;
                END_IF;
                IF _retval = WORD#8091 THEN
                    Messenger.Activate(UINT#1341,eAxoMessageCategory#Error);
                    Status.Error.Id := UINT#1341;
                    RETURN;
                END_IF;
                IF _retval = WORD#8094 THEN
                    Messenger.Activate(UINT#1342,eAxoMessageCategory#Error);
                    Status.Error.Id := UINT#1342;
                    RETURN;
                END_IF;
                IF _retval = WORD#8095 THEN
                    Messenger.Activate(UINT#1343,eAxoMessageCategory#Error);
                    Status.Error.Id := UINT#1343;
                    RETURN;
                END_IF;
                IF _retval = WORD#8096 THEN
                    Messenger.Activate(UINT#1344,eAxoMessageCategory#Error);
                    Status.Error.Id := UINT#1344;
                    RETURN;
                END_IF;
                IF _retval = WORD#8097 THEN
                    Messenger.Activate(UINT#1345,eAxoMessageCategory#Error);
                    Status.Error.Id := UINT#1345;
                    RETURN;
                END_IF;
                ReadHardwareIOAddress(hardwareID := (Config.HWIDs.HwID_ToolResult_58) , inputStartAddress => _inputsAddress , inputCount => _inputsCount , outputStartAddress => _outputsAddress , outputCount => _outputsCount);
                IF _inputsCount <> UINT#20 OR _outputsCount <> UINT#0 THEN
                    Messenger.Activate(UINT#1346,eAxoMessageCategory#Error);
                    Status.Error.Id := UINT#1346;
                    RETURN;
                END_IF;
                //******************Slot 65*****************//
                _geoAddr.Slot   :=  UINT#65;
                _geoAddr.HardwareType := UINT#4; // (4-Module)
                _retval := ReadHardwareIDFromSlot(geoAddr := _geoAddr, hardwareID => Config.HWIDs.HwID_ToolResult_59);
                IF Config.HWIDs.HwID_ToolResult_59 = UINT#0 THEN
                    Messenger.Activate(UINT#1350,eAxoMessageCategory#Error);
                    Status.Error.Id := UINT#1350;
                    RETURN;
                END_IF;
                IF _retval = WORD#8091 THEN
                    Messenger.Activate(UINT#1351,eAxoMessageCategory#Error);
                    Status.Error.Id := UINT#1351;
                    RETURN;
                END_IF;
                IF _retval = WORD#8094 THEN
                    Messenger.Activate(UINT#1352,eAxoMessageCategory#Error);
                    Status.Error.Id := UINT#1352;
                    RETURN;
                END_IF;
                IF _retval = WORD#8095 THEN
                    Messenger.Activate(UINT#1353,eAxoMessageCategory#Error);
                    Status.Error.Id := UINT#1353;
                    RETURN;
                END_IF;
                IF _retval = WORD#8096 THEN
                    Messenger.Activate(UINT#1354,eAxoMessageCategory#Error);
                    Status.Error.Id := UINT#1354;
                    RETURN;
                END_IF;
                IF _retval = WORD#8097 THEN
                    Messenger.Activate(UINT#1355,eAxoMessageCategory#Error);
                    Status.Error.Id := UINT#1355;
                    RETURN;
                END_IF;
                ReadHardwareIOAddress(hardwareID := (Config.HWIDs.HwID_ToolResult_59) , inputStartAddress => _inputsAddress , inputCount => _inputsCount , outputStartAddress => _outputsAddress , outputCount => _outputsCount);
                IF _inputsCount <> UINT#20 OR _outputsCount <> UINT#0 THEN
                    Messenger.Activate(UINT#1356,eAxoMessageCategory#Error);
                    Status.Error.Id := UINT#1356;
                    RETURN;
                END_IF;
                //******************Slot 66*****************//
                _geoAddr.Slot   :=  UINT#66;
                _geoAddr.HardwareType := UINT#4; // (4-Module)
                _retval := ReadHardwareIDFromSlot(geoAddr := _geoAddr, hardwareID => Config.HWIDs.HwID_ToolResult_60);
                IF Config.HWIDs.HwID_ToolResult_60 = UINT#0 THEN
                    Messenger.Activate(UINT#1360,eAxoMessageCategory#Error);
                    Status.Error.Id := UINT#1360;
                    RETURN;
                END_IF;
                IF _retval = WORD#8091 THEN
                    Messenger.Activate(UINT#1361,eAxoMessageCategory#Error);
                    Status.Error.Id := UINT#1361;
                    RETURN;
                END_IF;
                IF _retval = WORD#8094 THEN
                    Messenger.Activate(UINT#1362,eAxoMessageCategory#Error);
                    Status.Error.Id := UINT#1362;
                    RETURN;
                END_IF;
                IF _retval = WORD#8095 THEN
                    Messenger.Activate(UINT#1363,eAxoMessageCategory#Error);
                    Status.Error.Id := UINT#1363;
                    RETURN;
                END_IF;
                IF _retval = WORD#8096 THEN
                    Messenger.Activate(UINT#1364,eAxoMessageCategory#Error);
                    Status.Error.Id := UINT#1364;
                    RETURN;
                END_IF;
                IF _retval = WORD#8097 THEN
                    Messenger.Activate(UINT#1365,eAxoMessageCategory#Error);
                    Status.Error.Id := UINT#1365;
                    RETURN;
                END_IF;
                ReadHardwareIOAddress(hardwareID := (Config.HWIDs.HwID_ToolResult_60) , inputStartAddress => _inputsAddress , inputCount => _inputsCount , outputStartAddress => _outputsAddress , outputCount => _outputsCount);
                IF _inputsCount <> UINT#20 OR _outputsCount <> UINT#0 THEN
                    Messenger.Activate(UINT#1366,eAxoMessageCategory#Error);
                    Status.Error.Id := UINT#1366;
                    RETURN;
                END_IF;
                //******************Slot 67*****************//
                _geoAddr.Slot   :=  UINT#67;
                _geoAddr.HardwareType := UINT#4; // (4-Module)
                _retval := ReadHardwareIDFromSlot(geoAddr := _geoAddr, hardwareID => Config.HWIDs.HwID_ToolResult_61);
                IF Config.HWIDs.HwID_ToolResult_61 = UINT#0 THEN
                    Messenger.Activate(UINT#1370,eAxoMessageCategory#Error);
                    Status.Error.Id := UINT#1370;
                    RETURN;
                END_IF;
                IF _retval = WORD#8091 THEN
                    Messenger.Activate(UINT#1371,eAxoMessageCategory#Error);
                    Status.Error.Id := UINT#1371;
                    RETURN;
                END_IF;
                IF _retval = WORD#8094 THEN
                    Messenger.Activate(UINT#1372,eAxoMessageCategory#Error);
                    Status.Error.Id := UINT#1372;
                    RETURN;
                END_IF;
                IF _retval = WORD#8095 THEN
                    Messenger.Activate(UINT#1373,eAxoMessageCategory#Error);
                    Status.Error.Id := UINT#1373;
                    RETURN;
                END_IF;
                IF _retval = WORD#8096 THEN
                    Messenger.Activate(UINT#1374,eAxoMessageCategory#Error);
                    Status.Error.Id := UINT#1374;
                    RETURN;
                END_IF;
                IF _retval = WORD#8097 THEN
                    Messenger.Activate(UINT#1375,eAxoMessageCategory#Error);
                    Status.Error.Id := UINT#1375;
                    RETURN;
                END_IF;
                ReadHardwareIOAddress(hardwareID := (Config.HWIDs.HwID_ToolResult_61) , inputStartAddress => _inputsAddress , inputCount => _inputsCount , outputStartAddress => _outputsAddress , outputCount => _outputsCount);
                IF _inputsCount <> UINT#20 OR _outputsCount <> UINT#0 THEN
                    Messenger.Activate(UINT#1376,eAxoMessageCategory#Error);
                    Status.Error.Id := UINT#1376;
                    RETURN;
                END_IF;
                //******************Slot 68*****************//
                _geoAddr.Slot   :=  UINT#68;
                _geoAddr.HardwareType := UINT#4; // (4-Module)
                _retval := ReadHardwareIDFromSlot(geoAddr := _geoAddr, hardwareID => Config.HWIDs.HwID_ToolResult_62);
                IF Config.HWIDs.HwID_ToolResult_62 = UINT#0 THEN
                    Messenger.Activate(UINT#1380,eAxoMessageCategory#Error);
                    Status.Error.Id := UINT#1380;
                    RETURN;
                END_IF;
                IF _retval = WORD#8091 THEN
                    Messenger.Activate(UINT#1381,eAxoMessageCategory#Error);
                    Status.Error.Id := UINT#1381;
                    RETURN;
                END_IF;
                IF _retval = WORD#8094 THEN
                    Messenger.Activate(UINT#1382,eAxoMessageCategory#Error);
                    Status.Error.Id := UINT#1382;
                    RETURN;
                END_IF;
                IF _retval = WORD#8095 THEN
                    Messenger.Activate(UINT#1383,eAxoMessageCategory#Error);
                    Status.Error.Id := UINT#1383;
                    RETURN;
                END_IF;
                IF _retval = WORD#8096 THEN
                    Messenger.Activate(UINT#1384,eAxoMessageCategory#Error);
                    Status.Error.Id := UINT#1384;
                    RETURN;
                END_IF;
                IF _retval = WORD#8097 THEN
                    Messenger.Activate(UINT#1385,eAxoMessageCategory#Error);
                    Status.Error.Id := UINT#1385;
                    RETURN;
                END_IF;
                ReadHardwareIOAddress(hardwareID := (Config.HWIDs.HwID_ToolResult_62) , inputStartAddress => _inputsAddress , inputCount => _inputsCount , outputStartAddress => _outputsAddress , outputCount => _outputsCount);
                IF _inputsCount <> UINT#20 OR _outputsCount <> UINT#0 THEN
                    Messenger.Activate(UINT#1386,eAxoMessageCategory#Error);
                    Status.Error.Id := UINT#1386;
                    RETURN;
                END_IF;
                //******************Slot 69*****************//
                _geoAddr.Slot   :=  UINT#69;
                _geoAddr.HardwareType := UINT#4; // (4-Module)
                _retval := ReadHardwareIDFromSlot(geoAddr := _geoAddr, hardwareID => Config.HWIDs.HwID_ToolResult_63);
                IF Config.HWIDs.HwID_ToolResult_63 = UINT#0 THEN
                    Messenger.Activate(UINT#1390,eAxoMessageCategory#Error);
                    Status.Error.Id := UINT#1390;
                    RETURN;
                END_IF;
                IF _retval = WORD#8091 THEN
                    Messenger.Activate(UINT#1391,eAxoMessageCategory#Error);
                    Status.Error.Id := UINT#1391;
                    RETURN;
                END_IF;
                IF _retval = WORD#8094 THEN
                    Messenger.Activate(UINT#1392,eAxoMessageCategory#Error);
                    Status.Error.Id := UINT#1392;
                    RETURN;
                END_IF;
                IF _retval = WORD#8095 THEN
                    Messenger.Activate(UINT#1393,eAxoMessageCategory#Error);
                    Status.Error.Id := UINT#1393;
                    RETURN;
                END_IF;
                IF _retval = WORD#8096 THEN
                    Messenger.Activate(UINT#1394,eAxoMessageCategory#Error);
                    Status.Error.Id := UINT#1394;
                    RETURN;
                END_IF;
                IF _retval = WORD#8097 THEN
                    Messenger.Activate(UINT#1395,eAxoMessageCategory#Error);
                    Status.Error.Id := UINT#1395;
                    RETURN;
                END_IF;
                ReadHardwareIOAddress(hardwareID := (Config.HWIDs.HwID_ToolResult_63) , inputStartAddress => _inputsAddress , inputCount => _inputsCount , outputStartAddress => _outputsAddress , outputCount => _outputsCount);
                IF _inputsCount <> UINT#20 OR _outputsCount <> UINT#0 THEN
                    Messenger.Activate(UINT#1396,eAxoMessageCategory#Error);
                    Status.Error.Id := UINT#1396;
                    RETURN;
                END_IF;
                //******************Slot 70*****************//
                _geoAddr.Slot   :=  UINT#70;
                _geoAddr.HardwareType := UINT#4; // (4-Module)
                _retval := ReadHardwareIDFromSlot(geoAddr := _geoAddr, hardwareID => Config.HWIDs.HwID_ToolResult_64);
                IF Config.HWIDs.HwID_ToolResult_64 = UINT#0 THEN
                    Messenger.Activate(UINT#1400,eAxoMessageCategory#Error);
                    Status.Error.Id := UINT#1400;
                    RETURN;
                END_IF;
                IF _retval = WORD#8091 THEN
                    Messenger.Activate(UINT#1401,eAxoMessageCategory#Error);
                    Status.Error.Id := UINT#1401;
                    RETURN;
                END_IF;
                IF _retval = WORD#8094 THEN
                    Messenger.Activate(UINT#1402,eAxoMessageCategory#Error);
                    Status.Error.Id := UINT#1402;
                    RETURN;
                END_IF;
                IF _retval = WORD#8095 THEN
                    Messenger.Activate(UINT#1403,eAxoMessageCategory#Error);
                    Status.Error.Id := UINT#1403;
                    RETURN;
                END_IF;
                IF _retval = WORD#8096 THEN
                    Messenger.Activate(UINT#1404,eAxoMessageCategory#Error);
                    Status.Error.Id := UINT#1404;
                    RETURN;
                END_IF;
                IF _retval = WORD#8097 THEN
                    Messenger.Activate(UINT#1405,eAxoMessageCategory#Error);
                    Status.Error.Id := UINT#1405;
                    RETURN;
                END_IF;
                ReadHardwareIOAddress(hardwareID := (Config.HWIDs.HwID_ToolResult_64) , inputStartAddress => _inputsAddress , inputCount => _inputsCount , outputStartAddress => _outputsAddress , outputCount => _outputsCount);
                IF _inputsCount <> UINT#20 OR _outputsCount <> UINT#0 THEN
                    Messenger.Activate(UINT#1406,eAxoMessageCategory#Error);
                    Status.Error.Id := UINT#1406;
                    RETURN;
                END_IF;
                //******************Slot 71*****************//
                _geoAddr.Slot   :=  UINT#71;
                _geoAddr.HardwareType := UINT#4; // (4-Module)
                _retval := ReadHardwareIDFromSlot(geoAddr := _geoAddr, hardwareID => Config.HWIDs.HwID_DeviceResultBits_2);
                IF Config.HWIDs.HwID_DeviceResultBits_2 = UINT#0 THEN
                    Messenger.Activate(UINT#1410,eAxoMessageCategory#Error);
                    Status.Error.Id := UINT#1410;
                    RETURN;
                END_IF;
                IF _retval = WORD#8091 THEN
                    Messenger.Activate(UINT#1411,eAxoMessageCategory#Error);
                    Status.Error.Id := UINT#1411;
                    RETURN;
                END_IF;
                IF _retval = WORD#8094 THEN
                    Messenger.Activate(UINT#1412,eAxoMessageCategory#Error);
                    Status.Error.Id := UINT#1412;
                    RETURN;
                END_IF;
                IF _retval = WORD#8095 THEN
                    Messenger.Activate(UINT#1413,eAxoMessageCategory#Error);
                    Status.Error.Id := UINT#1413;
                    RETURN;
                END_IF;
                IF _retval = WORD#8096 THEN
                    Messenger.Activate(UINT#1414,eAxoMessageCategory#Error);
                    Status.Error.Id := UINT#1414;
                    RETURN;
                END_IF;
                IF _retval = WORD#8097 THEN
                    Messenger.Activate(UINT#1415,eAxoMessageCategory#Error);
                    Status.Error.Id := UINT#1415;
                    RETURN;
                END_IF;
                ReadHardwareIOAddress(hardwareID := (Config.HWIDs.HwID_DeviceResultBits_2) , inputStartAddress => _inputsAddress , inputCount => _inputsCount , outputStartAddress => _outputsAddress , outputCount => _outputsCount);
                IF _inputsCount <> UINT#8 OR _outputsCount <> UINT#0 THEN
                    Messenger.Activate(UINT#1416,eAxoMessageCategory#Error);
                    Status.Error.Id := UINT#1416;
                    RETURN;
                END_IF;
